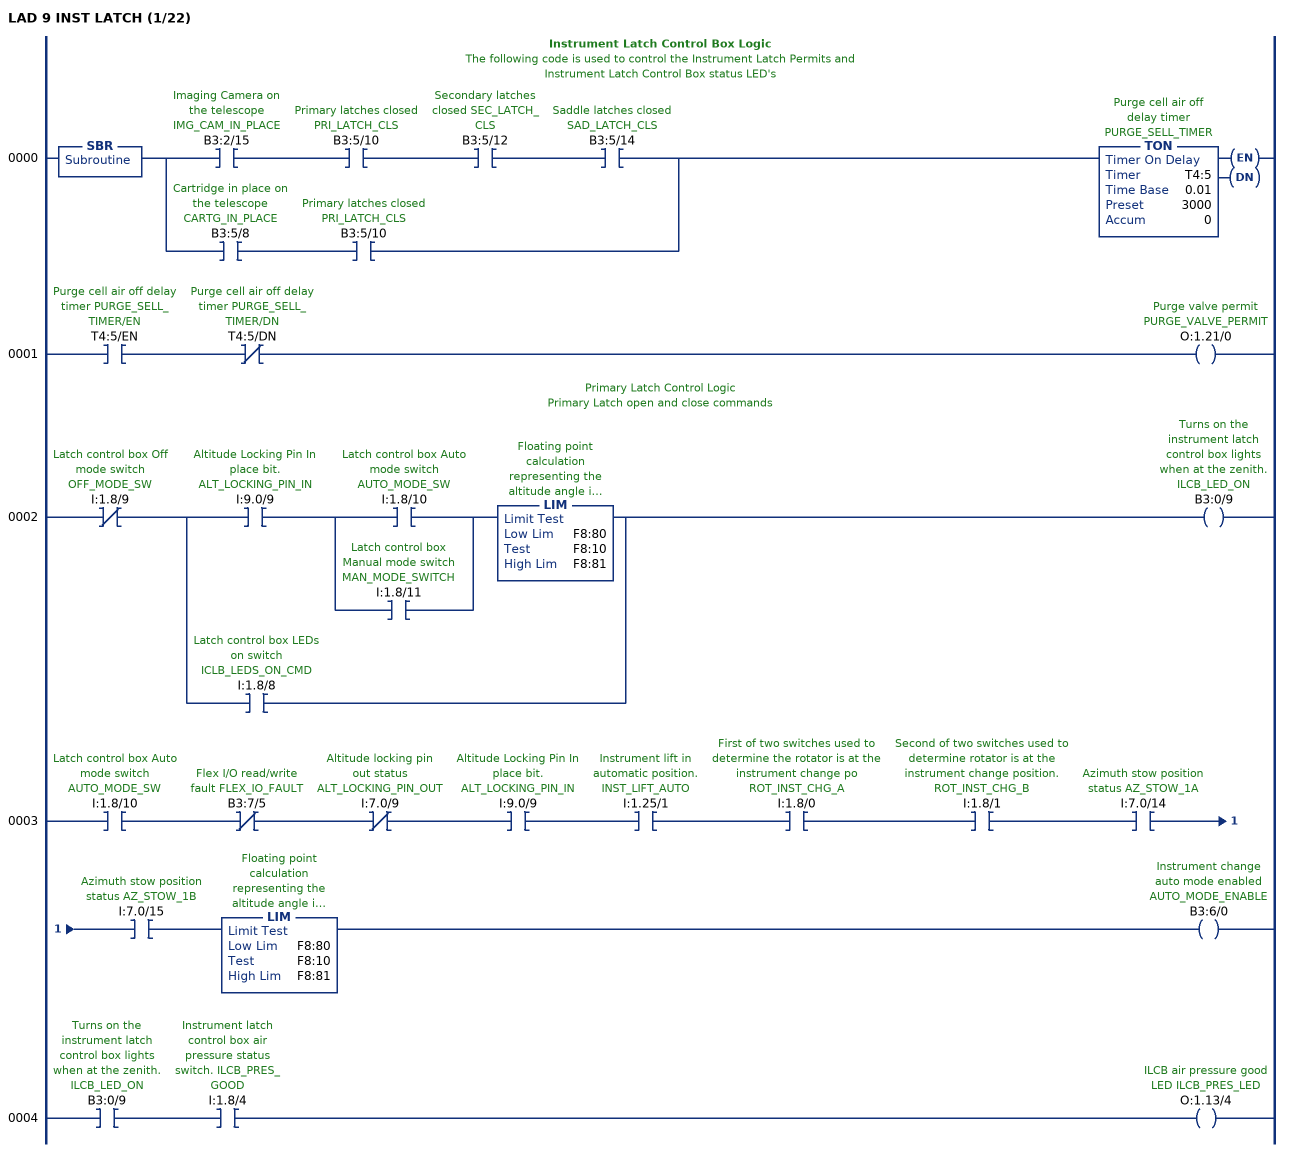
% Rung: 0 %
% TITLE: Instrument Latch Control Box Logic %
% The following code is used to control the Instrument Latch Permits and
% Instrument Latch Control Box status LED's %
SOR SBR BST XIC B3:2/15 XIC B3:5/10 XIC B3:5/12 XIC B3:5/14 NXB XIC B3:5/8 XIC B3:5/10 BND TON T4:5 0.01 3000 0 EOR
%   B3:2/15  IMG_CAM_IN_PLACE  "Imaging Camera on the telescope" %
%   B3:5/10  PRI_LATCH_CLS  "Primary latches closed" %
%   B3:5/12  SEC_LATCH_CLS  "Secondary latches closed" %
%   B3:5/14  SAD_LATCH_CLS  "Saddle latches closed" %
%   B3:5/8  CARTG_IN_PLACE  "Cartridge in place on the telescope" %
%   T4:5  PURGE_SELL_TIMER  "Purge cell air off delay timer" %
% Rung: 1 %
SOR XIC T4:5/EN XIO T4:5/DN OTE O:1.21/0 EOR
%   T4:5  PURGE_SELL_TIMER  "Purge cell air off delay timer" %
%   O:1.21/0  PURGE_VALVE_PERMIT  "Purge valve permit" %
% Rung: 2 %
% Primary Latch Control Logic
% 
% 
% 
% Primary Latch open and close commands %
SOR XIO I:1.8/9 BST XIC I:9.0/9 BST XIC I:1.8/10 NXB XIC I:1.8/11 BND LIM F8:80 F8:10 F8:81 NXB XIC I:1.8/8 BND OTE B3:0/9 EOR
%   I:1.8/9  OFF_MODE_SW  "Latch control box Off mode switch" %
%   I:9.0/9  ALT_LOCKING_PIN_IN  "Altitude Locking Pin In place bit." %
%   I:1.8/10  AUTO_MODE_SW  "Latch control box Auto mode switch" %
%   I:1.8/11  MAN_MODE_SWITCH  "Latch control box Manual mode switch" %
%   F8:80  INST_CHG_LOW_LMT  "The Lower altitude limit to allow instrument change operations" %
%   F8:10  ALT_ANGLE  "Floating point calculation representing the altitude angle in degrees." %
%   F8:81  INST_CHG_HIGH_LMT  "The Upper altitude limit to allow instrument change operations" %
%   I:1.8/8  ICLB_LEDS_ON_CMD  "Latch control box LEDs on switch" %
%   B3:0/9  ILCB_LED_ON  "Turns on the instrument latch control box lights when at the zenith." %
% Rung: 3 %
SOR XIC I:1.8/10 XIO B3:7/5 XIO I:7.0/9 XIC I:9.0/9 XIC I:1.25/1 XIC I:1.8/0 XIC I:1.8/1 XIC I:7.0/14 XIC I:7.0/15 LIM F8:80 F8:10 F8:81 OTE B3:6/0 EOR
%   I:1.8/10  AUTO_MODE_SW  "Latch control box Auto mode switch" %
%   B3:7/5  FLEX_IO_FAULT  "Flex I/O read/write fault" %
%   I:7.0/9  ALT_LOCKING_PIN_OUT  "Altitude locking pin out status" %
%   I:9.0/9  ALT_LOCKING_PIN_IN  "Altitude Locking Pin In place bit." %
%   I:1.25/1  INST_LIFT_AUTO  "Instrument lift in automatic position." %
%   I:1.8/0  ROT_INST_CHG_A  "First of two switches used to determine the rotator is at the instrument change po" %
%   I:1.8/1  ROT_INST_CHG_B  "Second of two switches used to determine rotator is at the instrument change position." %
%   I:7.0/14  AZ_STOW_1A  "Azimuth stow position status" %
%   I:7.0/15  AZ_STOW_1B  "Azimuth stow position status" %
%   F8:80  INST_CHG_LOW_LMT  "The Lower altitude limit to allow instrument change operations" %
%   F8:10  ALT_ANGLE  "Floating point calculation representing the altitude angle in degrees." %
%   F8:81  INST_CHG_HIGH_LMT  "The Upper altitude limit to allow instrument change operations" %
%   B3:6/0  AUTO_MODE_ENABLE  "Instrument change auto mode enabled" %
% Rung: 4 %
SOR XIC B3:0/9 XIC I:1.8/4 OTE O:1.13/4 EOR
%   B3:0/9  ILCB_LED_ON  "Turns on the instrument latch control box lights when at the zenith." %
%   I:1.8/4  ILCB_PRES_GOOD  "Instrument latch control box air pressure status switch." %
%   O:1.13/4  ILCB_PRES_LED  "ILCB air pressure good LED" %

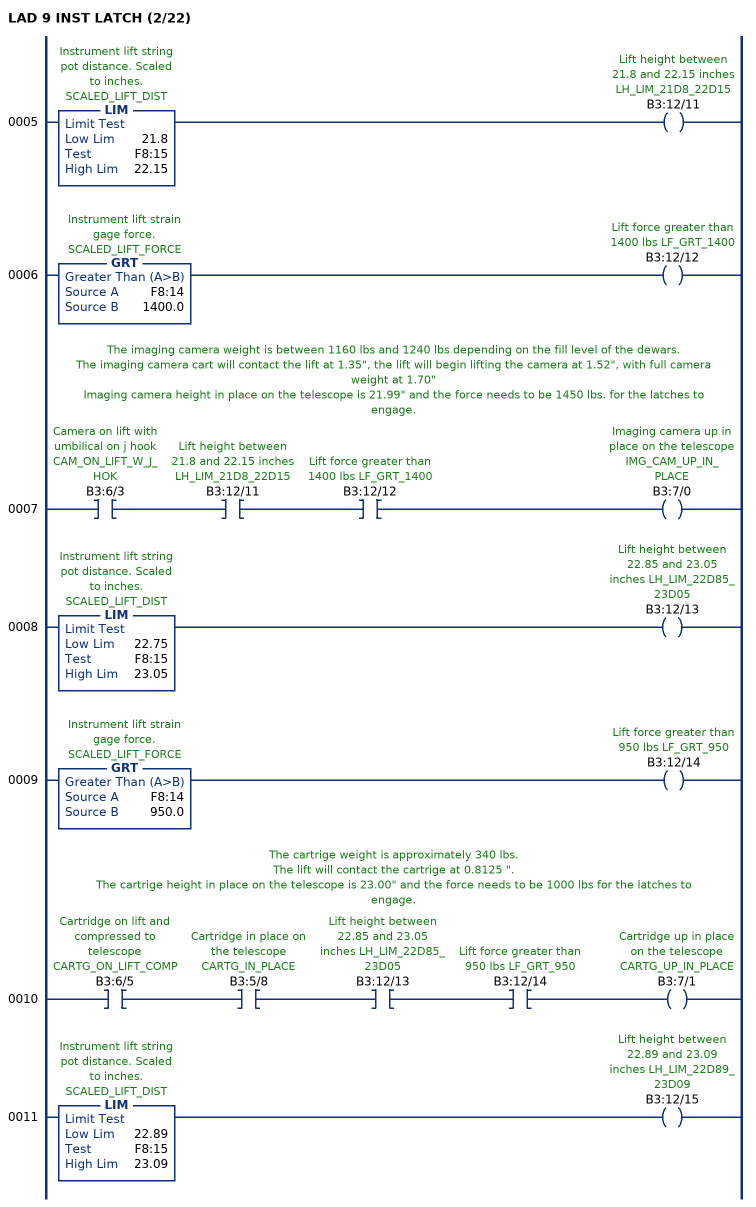
% Rung: 5 %
SOR LIM 21.8 F8:15 22.15 OTE B3:12/11 EOR
%   F8:15  SCALED_LIFT_DIST  "Instrument lift string pot distance. Scaled to inches." %
%   B3:12/11  LH_LIM_21D8_22D15  "Lift height between 21.8 and 22.15 inches" %
% Rung: 6 %
SOR GRT F8:14 1400.0 OTE B3:12/12 EOR
%   F8:14  SCALED_LIFT_FORCE  "Instrument lift strain gage force." %
%   B3:12/12  LF_GRT_1400  "Lift force greater than 1400 lbs" %
% Rung: 7 %
% The imaging camera weight is between 1160 lbs and 1240 lbs depending on the fill level of the dewars.
% The imaging camera cart will contact the lift at 1.35", the lift will begin lifting the camera at 1.52", with full camera weight at 1.70"
% Imaging camera height in place on the telescope is 21.99" and the force needs to be 1450 lbs. for the latches to engage. %
SOR XIC B3:6/3 XIC B3:12/11 XIC B3:12/12 OTE B3:7/0 EOR
%   B3:6/3  CAM_ON_LIFT_W_J_HOK  "Camera on lift with umbilical on j hook" %
%   B3:12/11  LH_LIM_21D8_22D15  "Lift height between 21.8 and 22.15 inches" %
%   B3:12/12  LF_GRT_1400  "Lift force greater than 1400 lbs" %
%   B3:7/0  IMG_CAM_UP_IN_PLACE  "Imaging camera up in place on the telescope" %
% Rung: 8 %
SOR LIM 22.75 F8:15 23.05 OTE B3:12/13 EOR
%   F8:15  SCALED_LIFT_DIST  "Instrument lift string pot distance. Scaled to inches." %
%   B3:12/13  LH_LIM_22D85_23D05  "Lift height between 22.85 and 23.05 inches" %
% Rung: 9 %
SOR GRT F8:14 950.0 OTE B3:12/14 EOR
%   F8:14  SCALED_LIFT_FORCE  "Instrument lift strain gage force." %
%   B3:12/14  LF_GRT_950  "Lift force greater than 950 lbs" %
% Rung: 10 %
% The cartrige weight is approximately 340 lbs.
% The lift will contact the cartrige at 0.8125 ".
% The cartrige height in place on the telescope is 23.00" and the force needs to be 1000 lbs for the latches to engage. %
SOR XIC B3:6/5 XIC B3:5/8 XIC B3:12/13 XIC B3:12/14 OTE B3:7/1 EOR
%   B3:6/5  CARTG_ON_LIFT_COMP  "Cartridge on lift and compressed to telescope" %
%   B3:5/8  CARTG_IN_PLACE  "Cartridge in place on the telescope" %
%   B3:12/13  LH_LIM_22D85_23D05  "Lift height between 22.85 and 23.05 inches" %
%   B3:12/14  LF_GRT_950  "Lift force greater than 950 lbs" %
%   B3:7/1  CARTG_UP_IN_PLACE  "Cartridge up in place on the telescope" %
% Rung: 11 %
SOR LIM 22.89 F8:15 23.09 OTE B3:12/15 EOR
%   F8:15  SCALED_LIFT_DIST  "Instrument lift string pot distance. Scaled to inches." %
%   B3:12/15  LH_LIM_22D89_23D09  "Lift height between 22.89 and 23.09 inches" %

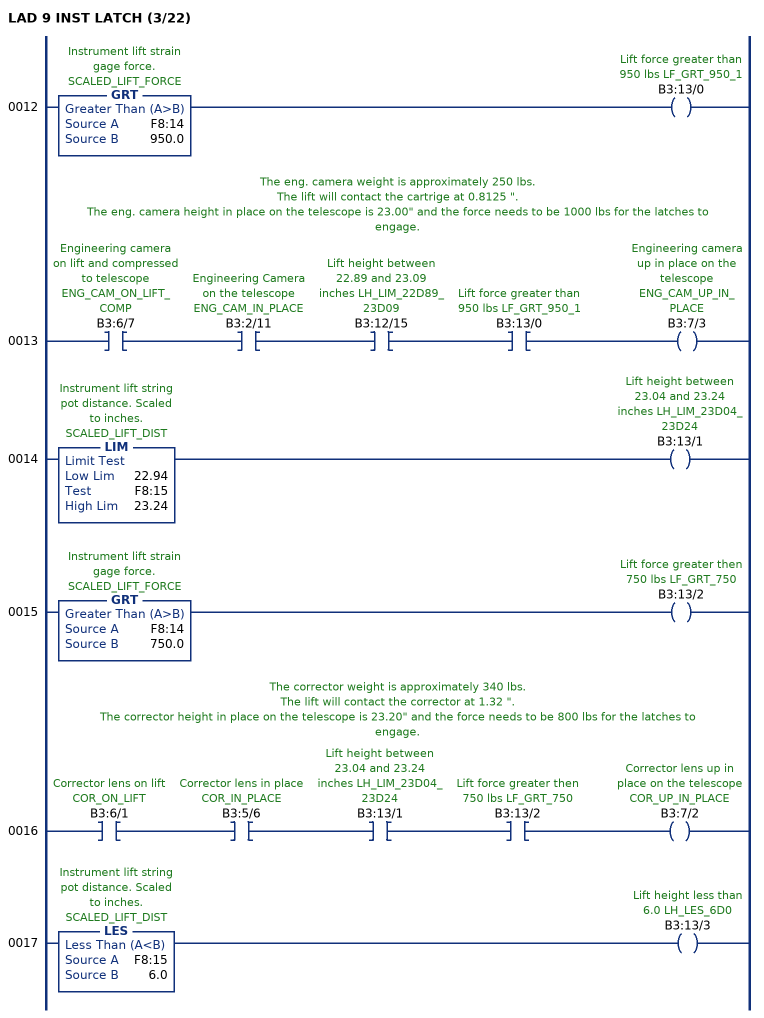
% Rung: 12 %
SOR GRT F8:14 950.0 OTE B3:13/0 EOR
%   F8:14  SCALED_LIFT_FORCE  "Instrument lift strain gage force." %
%   B3:13/0  LF_GRT_950_1  "Lift force greater than 950 lbs" %
% Rung: 13 %
% The eng. camera weight is approximately 250 lbs.
% The lift will contact the cartrige at 0.8125 ".
% The eng. camera height in place on the telescope is 23.00" and the force needs to be 1000 lbs for the latches to engage. %
SOR XIC B3:6/7 XIC B3:2/11 XIC B3:12/15 XIC B3:13/0 OTE B3:7/3 EOR
%   B3:6/7  ENG_CAM_ON_LIFT_COMP  "Engineering camera on lift and compressed to telescope" %
%   B3:2/11  ENG_CAM_IN_PLACE  "Engineering Camera on the telescope" %
%   B3:12/15  LH_LIM_22D89_23D09  "Lift height between 22.89 and 23.09 inches" %
%   B3:13/0  LF_GRT_950_1  "Lift force greater than 950 lbs" %
%   B3:7/3  ENG_CAM_UP_IN_PLACE  "Engineering camera up in place on the telescope" %
% Rung: 14 %
SOR LIM 22.94 F8:15 23.24 OTE B3:13/1 EOR
%   F8:15  SCALED_LIFT_DIST  "Instrument lift string pot distance. Scaled to inches." %
%   B3:13/1  LH_LIM_23D04_23D24  "Lift height between 23.04 and 23.24 inches" %
% Rung: 15 %
SOR GRT F8:14 750.0 OTE B3:13/2 EOR
%   F8:14  SCALED_LIFT_FORCE  "Instrument lift strain gage force." %
%   B3:13/2  LF_GRT_750  "Lift force greater then 750 lbs" %
% Rung: 16 %
% The corrector weight is approximately 340 lbs.
% The lift will contact the corrector at 1.32 ".
% The corrector height in place on the telescope is 23.20" and the force needs to be 800 lbs for the latches to engage. %
SOR XIC B3:6/1 XIC B3:5/6 XIC B3:13/1 XIC B3:13/2 OTE B3:7/2 EOR
%   B3:6/1  COR_ON_LIFT  "Corrector lens on lift" %
%   B3:5/6  COR_IN_PLACE  "Corrector lens in place" %
%   B3:13/1  LH_LIM_23D04_23D24  "Lift height between 23.04 and 23.24 inches" %
%   B3:13/2  LF_GRT_750  "Lift force greater then 750 lbs" %
%   B3:7/2  COR_UP_IN_PLACE  "Corrector lens up in place on the telescope" %
% Rung: 17 %
SOR LES F8:15 6.0 OTE B3:13/3 EOR
%   F8:15  SCALED_LIFT_DIST  "Instrument lift string pot distance. Scaled to inches." %
%   B3:13/3  LH_LES_6D0  "Lift height less than 6.0" %

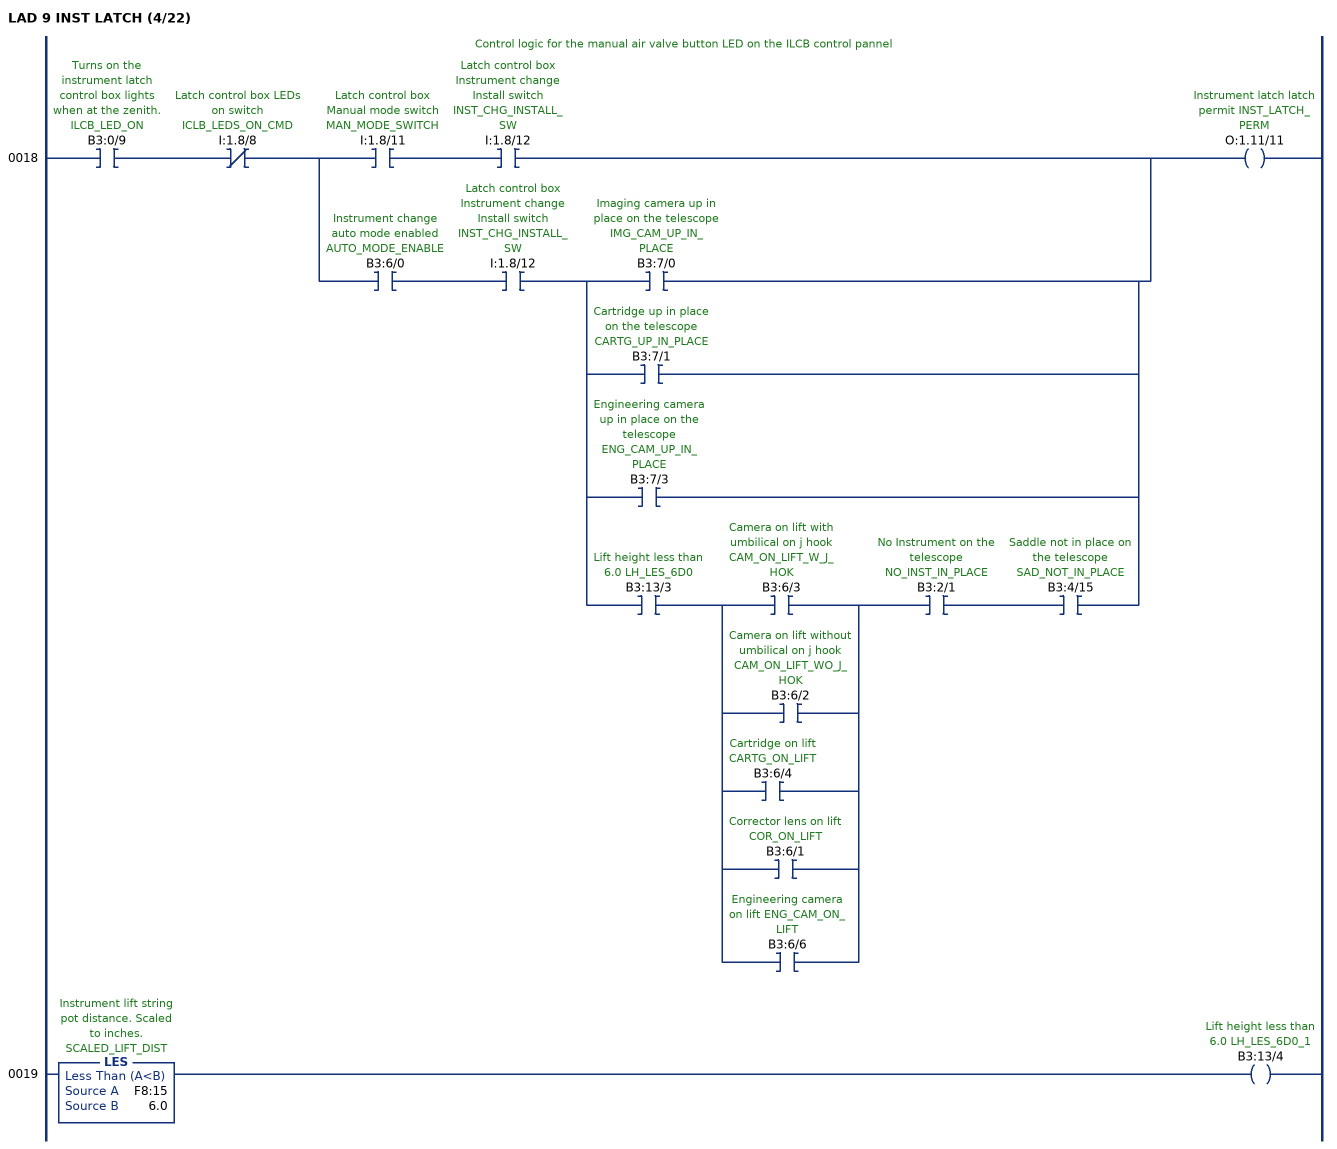
% Rung: 18 %
% Control logic for the manual air valve button LED on the ILCB control pannel %
SOR XIC B3:0/9 XIO I:1.8/8 BST XIC I:1.8/11 XIC I:1.8/12 NXB XIC B3:6/0 XIC I:1.8/12 BST XIC B3:7/0 NXB XIC B3:7/1 NXB XIC B3:7/3 NXB XIC B3:13/3 BST XIC B3:6/3 NXB XIC B3:6/2 NXB XIC B3:6/4 NXB XIC B3:6/1 NXB XIC B3:6/6 BND XIC B3:2/1 XIC B3:4/15 BND BND OTE O:1.11/11 EOR
%   B3:0/9  ILCB_LED_ON  "Turns on the instrument latch control box lights when at the zenith." %
%   I:1.8/8  ICLB_LEDS_ON_CMD  "Latch control box LEDs on switch" %
%   I:1.8/11  MAN_MODE_SWITCH  "Latch control box Manual mode switch" %
%   I:1.8/12  INST_CHG_INSTALL_SW  "Latch control box Instrument change Install switch" %
%   B3:6/0  AUTO_MODE_ENABLE  "Instrument change auto mode enabled" %
%   B3:7/0  IMG_CAM_UP_IN_PLACE  "Imaging camera up in place on the telescope" %
%   B3:7/1  CARTG_UP_IN_PLACE  "Cartridge up in place on the telescope" %
%   B3:7/3  ENG_CAM_UP_IN_PLACE  "Engineering camera up in place on the telescope" %
%   B3:13/3  LH_LES_6D0  "Lift height less than 6.0" %
%   B3:6/3  CAM_ON_LIFT_W_J_HOK  "Camera on lift with umbilical on j hook" %
%   B3:6/2  CAM_ON_LIFT_WO_J_HOK  "Camera on lift without umbilical on j hook" %
%   B3:6/4  CARTG_ON_LIFT  "Cartridge on lift" %
%   B3:6/1  COR_ON_LIFT  "Corrector lens on lift" %
%   B3:6/6  ENG_CAM_ON_LIFT  "Engineering camera on lift" %
%   B3:2/1  NO_INST_IN_PLACE  "No Instrument on the telescope" %
%   B3:4/15  SAD_NOT_IN_PLACE  "Saddle not in place on the telescope" %
%   O:1.11/11  INST_LATCH_PERM  "Instrument latch latch permit" %
% Rung: 19 %
SOR LES F8:15 6.0 OTE B3:13/4 EOR
%   F8:15  SCALED_LIFT_DIST  "Instrument lift string pot distance. Scaled to inches." %
%   B3:13/4  LH_LES_6D0_1  "Lift height less than 6.0" %

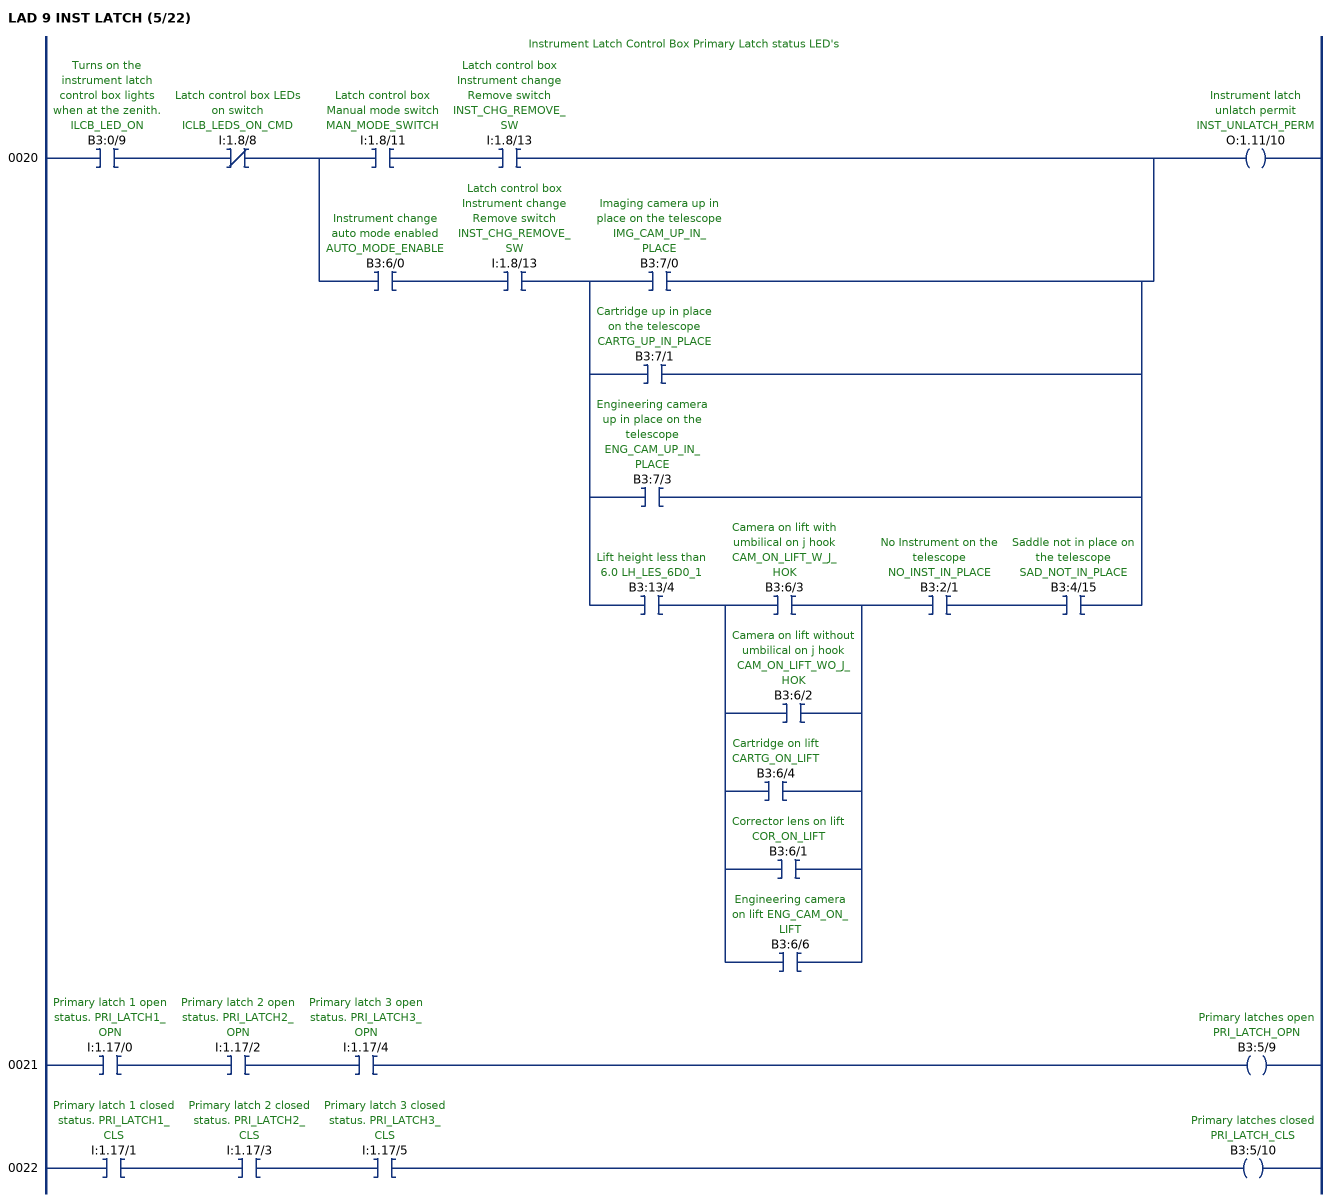
% Rung: 20 %
% Instrument Latch Control Box Primary Latch status LED's %
SOR XIC B3:0/9 XIO I:1.8/8 BST XIC I:1.8/11 XIC I:1.8/13 NXB XIC B3:6/0 XIC I:1.8/13 BST XIC B3:7/0 NXB XIC B3:7/1 NXB XIC B3:7/3 NXB XIC B3:13/4 BST XIC B3:6/3 NXB XIC B3:6/2 NXB XIC B3:6/4 NXB XIC B3:6/1 NXB XIC B3:6/6 BND XIC B3:2/1 XIC B3:4/15 BND BND OTE O:1.11/10 EOR
%   B3:0/9  ILCB_LED_ON  "Turns on the instrument latch control box lights when at the zenith." %
%   I:1.8/8  ICLB_LEDS_ON_CMD  "Latch control box LEDs on switch" %
%   I:1.8/11  MAN_MODE_SWITCH  "Latch control box Manual mode switch" %
%   I:1.8/13  INST_CHG_REMOVE_SW  "Latch control box Instrument change Remove switch" %
%   B3:6/0  AUTO_MODE_ENABLE  "Instrument change auto mode enabled" %
%   B3:7/0  IMG_CAM_UP_IN_PLACE  "Imaging camera up in place on the telescope" %
%   B3:7/1  CARTG_UP_IN_PLACE  "Cartridge up in place on the telescope" %
%   B3:7/3  ENG_CAM_UP_IN_PLACE  "Engineering camera up in place on the telescope" %
%   B3:13/4  LH_LES_6D0_1  "Lift height less than 6.0" %
%   B3:6/3  CAM_ON_LIFT_W_J_HOK  "Camera on lift with umbilical on j hook" %
%   B3:6/2  CAM_ON_LIFT_WO_J_HOK  "Camera on lift without umbilical on j hook" %
%   B3:6/4  CARTG_ON_LIFT  "Cartridge on lift" %
%   B3:6/1  COR_ON_LIFT  "Corrector lens on lift" %
%   B3:6/6  ENG_CAM_ON_LIFT  "Engineering camera on lift" %
%   B3:2/1  NO_INST_IN_PLACE  "No Instrument on the telescope" %
%   B3:4/15  SAD_NOT_IN_PLACE  "Saddle not in place on the telescope" %
%   O:1.11/10  INST_UNLATCH_PERM  "Instrument latch unlatch permit" %
% Rung: 21 %
SOR XIC I:1.17/0 XIC I:1.17/2 XIC I:1.17/4 OTE B3:5/9 EOR
%   I:1.17/0  PRI_LATCH1_OPN  "Primary latch 1 open status." %
%   I:1.17/2  PRI_LATCH2_OPN  "Primary latch 2 open status." %
%   I:1.17/4  PRI_LATCH3_OPN  "Primary latch 3 open status." %
%   B3:5/9  PRI_LATCH_OPN  "Primary latches open" %
% Rung: 22 %
SOR XIC I:1.17/1 XIC I:1.17/3 XIC I:1.17/5 OTE B3:5/10 EOR
%   I:1.17/1  PRI_LATCH1_CLS  "Primary latch 1 closed status." %
%   I:1.17/3  PRI_LATCH2_CLS  "Primary latch 2 closed status." %
%   I:1.17/5  PRI_LATCH3_CLS  "Primary latch 3 closed status." %
%   B3:5/10  PRI_LATCH_CLS  "Primary latches closed" %

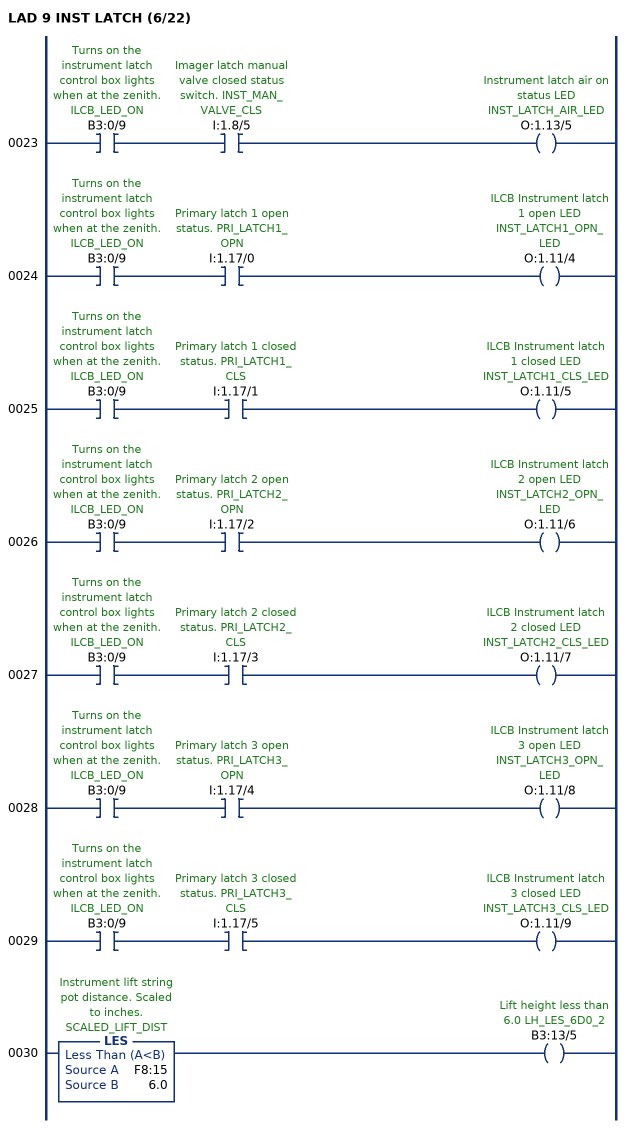
% Rung: 23 %
SOR XIC B3:0/9 XIC I:1.8/5 OTE O:1.13/5 EOR
%   B3:0/9  ILCB_LED_ON  "Turns on the instrument latch control box lights when at the zenith." %
%   I:1.8/5  INST_MAN_VALVE_CLS  "Imager latch manual valve closed status switch." %
%   O:1.13/5  INST_LATCH_AIR_LED  "Instrument latch air on status LED" %
% Rung: 24 %
SOR XIC B3:0/9 XIC I:1.17/0 OTE O:1.11/4 EOR
%   B3:0/9  ILCB_LED_ON  "Turns on the instrument latch control box lights when at the zenith." %
%   I:1.17/0  PRI_LATCH1_OPN  "Primary latch 1 open status." %
%   O:1.11/4  INST_LATCH1_OPN_LED  "ILCB Instrument latch 1 open LED" %
% Rung: 25 %
SOR XIC B3:0/9 XIC I:1.17/1 OTE O:1.11/5 EOR
%   B3:0/9  ILCB_LED_ON  "Turns on the instrument latch control box lights when at the zenith." %
%   I:1.17/1  PRI_LATCH1_CLS  "Primary latch 1 closed status." %
%   O:1.11/5  INST_LATCH1_CLS_LED  "ILCB Instrument latch 1 closed LED" %
% Rung: 26 %
SOR XIC B3:0/9 XIC I:1.17/2 OTE O:1.11/6 EOR
%   B3:0/9  ILCB_LED_ON  "Turns on the instrument latch control box lights when at the zenith." %
%   I:1.17/2  PRI_LATCH2_OPN  "Primary latch 2 open status." %
%   O:1.11/6  INST_LATCH2_OPN_LED  "ILCB Instrument latch 2 open LED" %
% Rung: 27 %
SOR XIC B3:0/9 XIC I:1.17/3 OTE O:1.11/7 EOR
%   B3:0/9  ILCB_LED_ON  "Turns on the instrument latch control box lights when at the zenith." %
%   I:1.17/3  PRI_LATCH2_CLS  "Primary latch 2 closed status." %
%   O:1.11/7  INST_LATCH2_CLS_LED  "ILCB Instrument latch 2 closed LED" %
% Rung: 28 %
SOR XIC B3:0/9 XIC I:1.17/4 OTE O:1.11/8 EOR
%   B3:0/9  ILCB_LED_ON  "Turns on the instrument latch control box lights when at the zenith." %
%   I:1.17/4  PRI_LATCH3_OPN  "Primary latch 3 open status." %
%   O:1.11/8  INST_LATCH3_OPN_LED  "ILCB Instrument latch 3 open LED" %
% Rung: 29 %
SOR XIC B3:0/9 XIC I:1.17/5 OTE O:1.11/9 EOR
%   B3:0/9  ILCB_LED_ON  "Turns on the instrument latch control box lights when at the zenith." %
%   I:1.17/5  PRI_LATCH3_CLS  "Primary latch 3 closed status." %
%   O:1.11/9  INST_LATCH3_CLS_LED  "ILCB Instrument latch 3 closed LED" %
% Rung: 30 %
SOR LES F8:15 6.0 OTE B3:13/5 EOR
%   F8:15  SCALED_LIFT_DIST  "Instrument lift string pot distance. Scaled to inches." %
%   B3:13/5  LH_LES_6D0_2  "Lift height less than 6.0" %

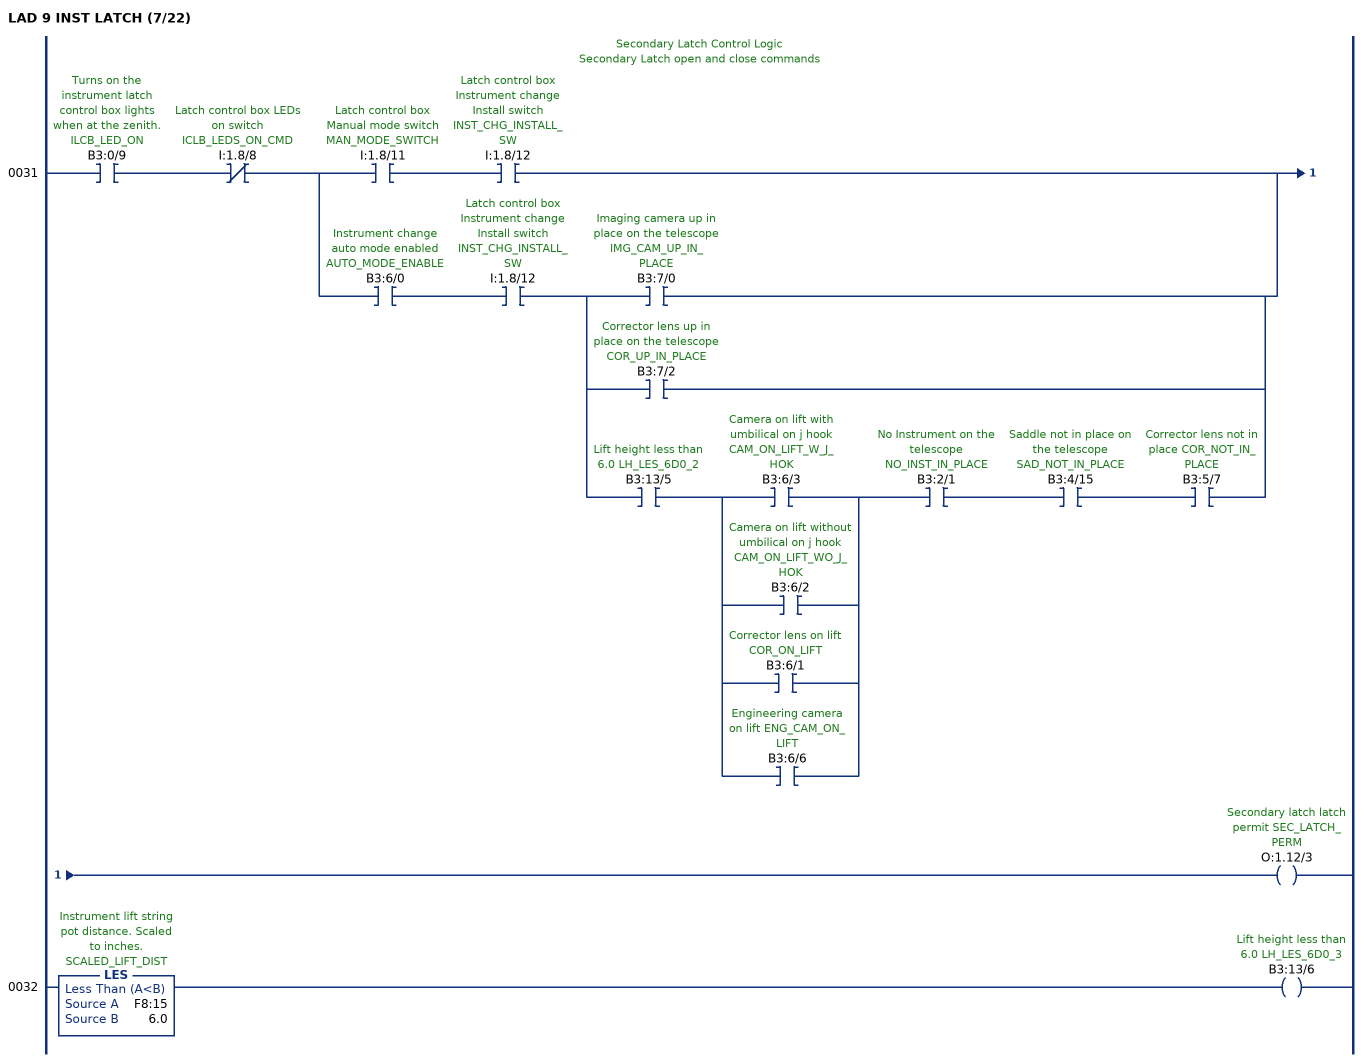
% Rung: 31 %
% Secondary Latch Control Logic
% 
% 
% 
% Secondary Latch open and close commands %
SOR XIC B3:0/9 XIO I:1.8/8 BST XIC I:1.8/11 XIC I:1.8/12 NXB XIC B3:6/0 XIC I:1.8/12 BST XIC B3:7/0 NXB XIC B3:7/2 NXB XIC B3:13/5 BST XIC B3:6/3 NXB XIC B3:6/2 NXB XIC B3:6/1 NXB XIC B3:6/6 BND XIC B3:2/1 XIC B3:4/15 XIC B3:5/7 BND BND OTE O:1.12/3 EOR
%   B3:0/9  ILCB_LED_ON  "Turns on the instrument latch control box lights when at the zenith." %
%   I:1.8/8  ICLB_LEDS_ON_CMD  "Latch control box LEDs on switch" %
%   I:1.8/11  MAN_MODE_SWITCH  "Latch control box Manual mode switch" %
%   I:1.8/12  INST_CHG_INSTALL_SW  "Latch control box Instrument change Install switch" %
%   B3:6/0  AUTO_MODE_ENABLE  "Instrument change auto mode enabled" %
%   B3:7/0  IMG_CAM_UP_IN_PLACE  "Imaging camera up in place on the telescope" %
%   B3:7/2  COR_UP_IN_PLACE  "Corrector lens up in place on the telescope" %
%   B3:13/5  LH_LES_6D0_2  "Lift height less than 6.0" %
%   B3:6/3  CAM_ON_LIFT_W_J_HOK  "Camera on lift with umbilical on j hook" %
%   B3:6/2  CAM_ON_LIFT_WO_J_HOK  "Camera on lift without umbilical on j hook" %
%   B3:6/1  COR_ON_LIFT  "Corrector lens on lift" %
%   B3:6/6  ENG_CAM_ON_LIFT  "Engineering camera on lift" %
%   B3:2/1  NO_INST_IN_PLACE  "No Instrument on the telescope" %
%   B3:4/15  SAD_NOT_IN_PLACE  "Saddle not in place on the telescope" %
%   B3:5/7  COR_NOT_IN_PLACE  "Corrector lens not in place" %
%   O:1.12/3  SEC_LATCH_PERM  "Secondary latch latch permit" %
% Rung: 32 %
SOR LES F8:15 6.0 OTE B3:13/6 EOR
%   F8:15  SCALED_LIFT_DIST  "Instrument lift string pot distance. Scaled to inches." %
%   B3:13/6  LH_LES_6D0_3  "Lift height less than 6.0" %

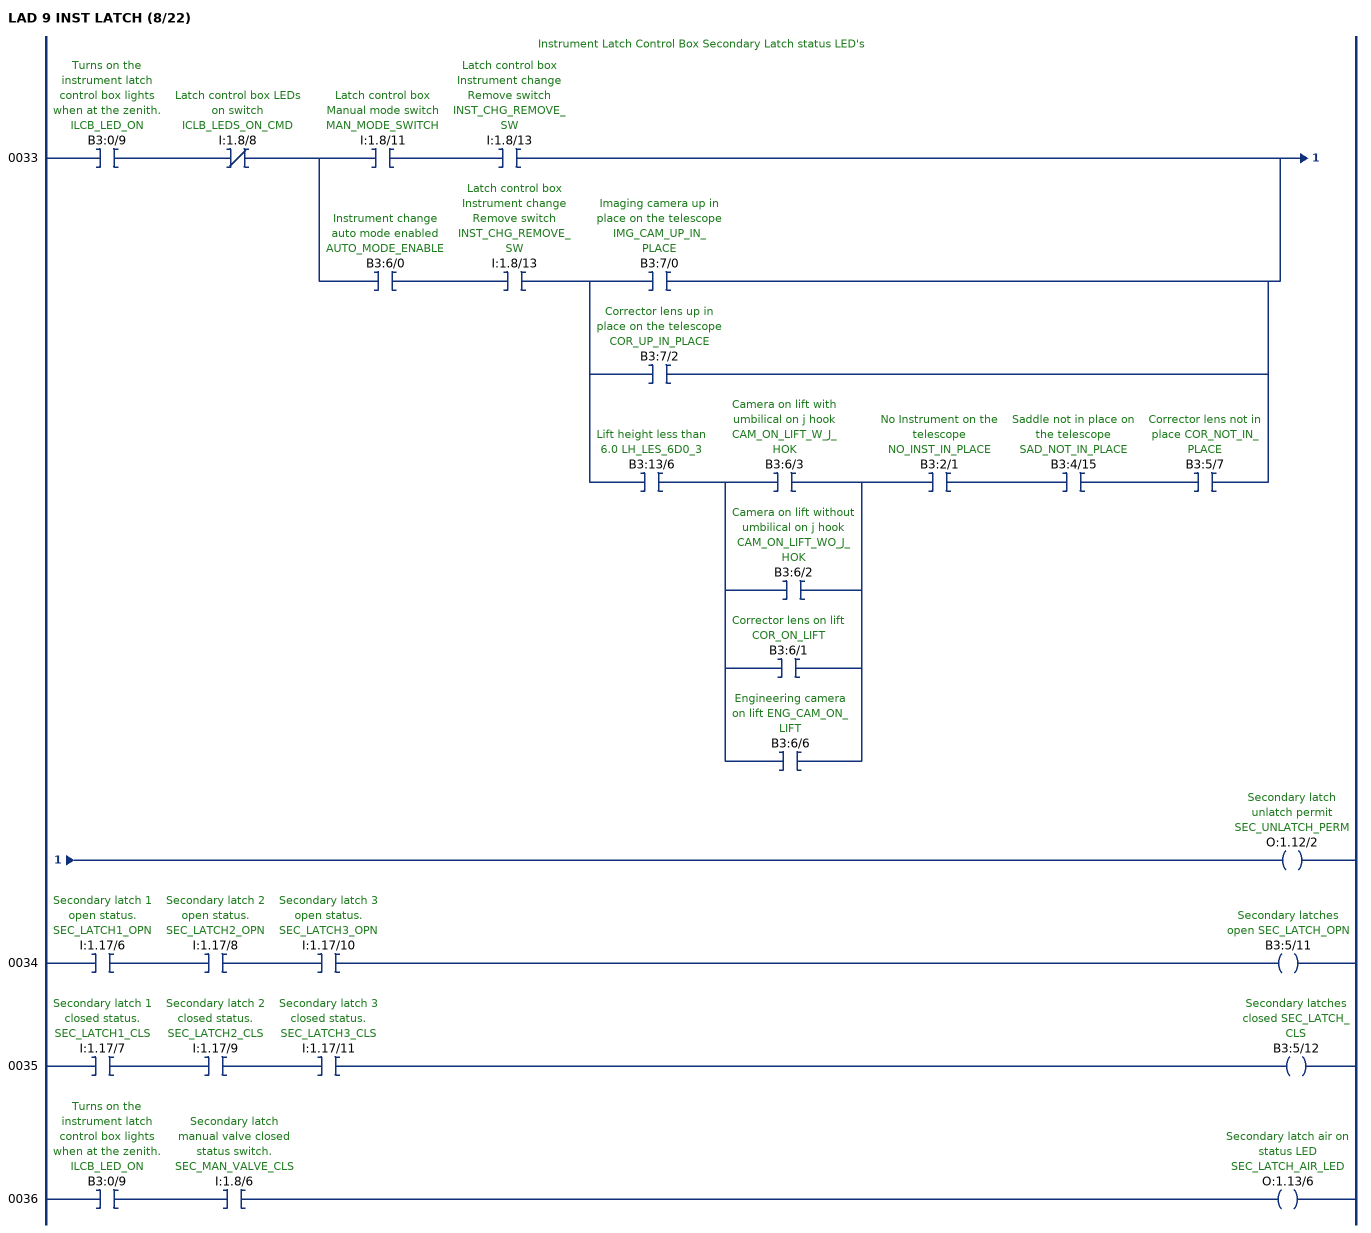
% Rung: 33 %
% Instrument Latch Control Box Secondary Latch status LED's %
SOR XIC B3:0/9 XIO I:1.8/8 BST XIC I:1.8/11 XIC I:1.8/13 NXB XIC B3:6/0 XIC I:1.8/13 BST XIC B3:7/0 NXB XIC B3:7/2 NXB XIC B3:13/6 BST XIC B3:6/3 NXB XIC B3:6/2 NXB XIC B3:6/1 NXB XIC B3:6/6 BND XIC B3:2/1 XIC B3:4/15 XIC B3:5/7 BND BND OTE O:1.12/2 EOR
%   B3:0/9  ILCB_LED_ON  "Turns on the instrument latch control box lights when at the zenith." %
%   I:1.8/8  ICLB_LEDS_ON_CMD  "Latch control box LEDs on switch" %
%   I:1.8/11  MAN_MODE_SWITCH  "Latch control box Manual mode switch" %
%   I:1.8/13  INST_CHG_REMOVE_SW  "Latch control box Instrument change Remove switch" %
%   B3:6/0  AUTO_MODE_ENABLE  "Instrument change auto mode enabled" %
%   B3:7/0  IMG_CAM_UP_IN_PLACE  "Imaging camera up in place on the telescope" %
%   B3:7/2  COR_UP_IN_PLACE  "Corrector lens up in place on the telescope" %
%   B3:13/6  LH_LES_6D0_3  "Lift height less than 6.0" %
%   B3:6/3  CAM_ON_LIFT_W_J_HOK  "Camera on lift with umbilical on j hook" %
%   B3:6/2  CAM_ON_LIFT_WO_J_HOK  "Camera on lift without umbilical on j hook" %
%   B3:6/1  COR_ON_LIFT  "Corrector lens on lift" %
%   B3:6/6  ENG_CAM_ON_LIFT  "Engineering camera on lift" %
%   B3:2/1  NO_INST_IN_PLACE  "No Instrument on the telescope" %
%   B3:4/15  SAD_NOT_IN_PLACE  "Saddle not in place on the telescope" %
%   B3:5/7  COR_NOT_IN_PLACE  "Corrector lens not in place" %
%   O:1.12/2  SEC_UNLATCH_PERM  "Secondary latch unlatch permit" %
% Rung: 34 %
SOR XIC I:1.17/6 XIC I:1.17/8 XIC I:1.17/10 OTE B3:5/11 EOR
%   I:1.17/6  SEC_LATCH1_OPN  "Secondary latch 1 open status." %
%   I:1.17/8  SEC_LATCH2_OPN  "Secondary latch 2 open status." %
%   I:1.17/10  SEC_LATCH3_OPN  "Secondary latch 3 open status." %
%   B3:5/11  SEC_LATCH_OPN  "Secondary latches open" %
% Rung: 35 %
SOR XIC I:1.17/7 XIC I:1.17/9 XIC I:1.17/11 OTE B3:5/12 EOR
%   I:1.17/7  SEC_LATCH1_CLS  "Secondary latch 1 closed status." %
%   I:1.17/9  SEC_LATCH2_CLS  "Secondary latch 2 closed status." %
%   I:1.17/11  SEC_LATCH3_CLS  "Secondary latch 3 closed status." %
%   B3:5/12  SEC_LATCH_CLS  "Secondary latches closed" %
% Rung: 36 %
SOR XIC B3:0/9 XIC I:1.8/6 OTE O:1.13/6 EOR
%   B3:0/9  ILCB_LED_ON  "Turns on the instrument latch control box lights when at the zenith." %
%   I:1.8/6  SEC_MAN_VALVE_CLS  "Secondary latch manual valve closed status switch." %
%   O:1.13/6  SEC_LATCH_AIR_LED  "Secondary latch air on status LED" %

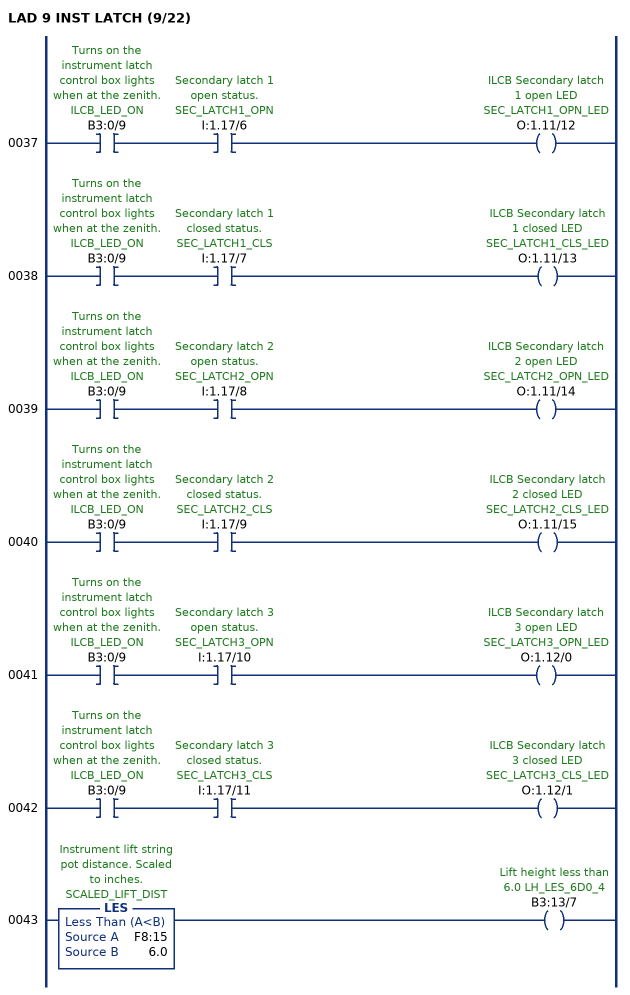
% Rung: 37 %
SOR XIC B3:0/9 XIC I:1.17/6 OTE O:1.11/12 EOR
%   B3:0/9  ILCB_LED_ON  "Turns on the instrument latch control box lights when at the zenith." %
%   I:1.17/6  SEC_LATCH1_OPN  "Secondary latch 1 open status." %
%   O:1.11/12  SEC_LATCH1_OPN_LED  "ILCB Secondary latch 1 open LED" %
% Rung: 38 %
SOR XIC B3:0/9 XIC I:1.17/7 OTE O:1.11/13 EOR
%   B3:0/9  ILCB_LED_ON  "Turns on the instrument latch control box lights when at the zenith." %
%   I:1.17/7  SEC_LATCH1_CLS  "Secondary latch 1 closed status." %
%   O:1.11/13  SEC_LATCH1_CLS_LED  "ILCB Secondary latch 1 closed LED" %
% Rung: 39 %
SOR XIC B3:0/9 XIC I:1.17/8 OTE O:1.11/14 EOR
%   B3:0/9  ILCB_LED_ON  "Turns on the instrument latch control box lights when at the zenith." %
%   I:1.17/8  SEC_LATCH2_OPN  "Secondary latch 2 open status." %
%   O:1.11/14  SEC_LATCH2_OPN_LED  "ILCB Secondary latch 2 open LED" %
% Rung: 40 %
SOR XIC B3:0/9 XIC I:1.17/9 OTE O:1.11/15 EOR
%   B3:0/9  ILCB_LED_ON  "Turns on the instrument latch control box lights when at the zenith." %
%   I:1.17/9  SEC_LATCH2_CLS  "Secondary latch 2 closed status." %
%   O:1.11/15  SEC_LATCH2_CLS_LED  "ILCB Secondary latch 2 closed LED" %
% Rung: 41 %
SOR XIC B3:0/9 XIC I:1.17/10 OTE O:1.12/0 EOR
%   B3:0/9  ILCB_LED_ON  "Turns on the instrument latch control box lights when at the zenith." %
%   I:1.17/10  SEC_LATCH3_OPN  "Secondary latch 3 open status." %
%   O:1.12/0  SEC_LATCH3_OPN_LED  "ILCB Secondary latch 3 open LED" %
% Rung: 42 %
SOR XIC B3:0/9 XIC I:1.17/11 OTE O:1.12/1 EOR
%   B3:0/9  ILCB_LED_ON  "Turns on the instrument latch control box lights when at the zenith." %
%   I:1.17/11  SEC_LATCH3_CLS  "Secondary latch 3 closed status." %
%   O:1.12/1  SEC_LATCH3_CLS_LED  "ILCB Secondary latch 3 closed LED" %
% Rung: 43 %
SOR LES F8:15 6.0 OTE B3:13/7 EOR
%   F8:15  SCALED_LIFT_DIST  "Instrument lift string pot distance. Scaled to inches." %
%   B3:13/7  LH_LES_6D0_4  "Lift height less than 6.0" %

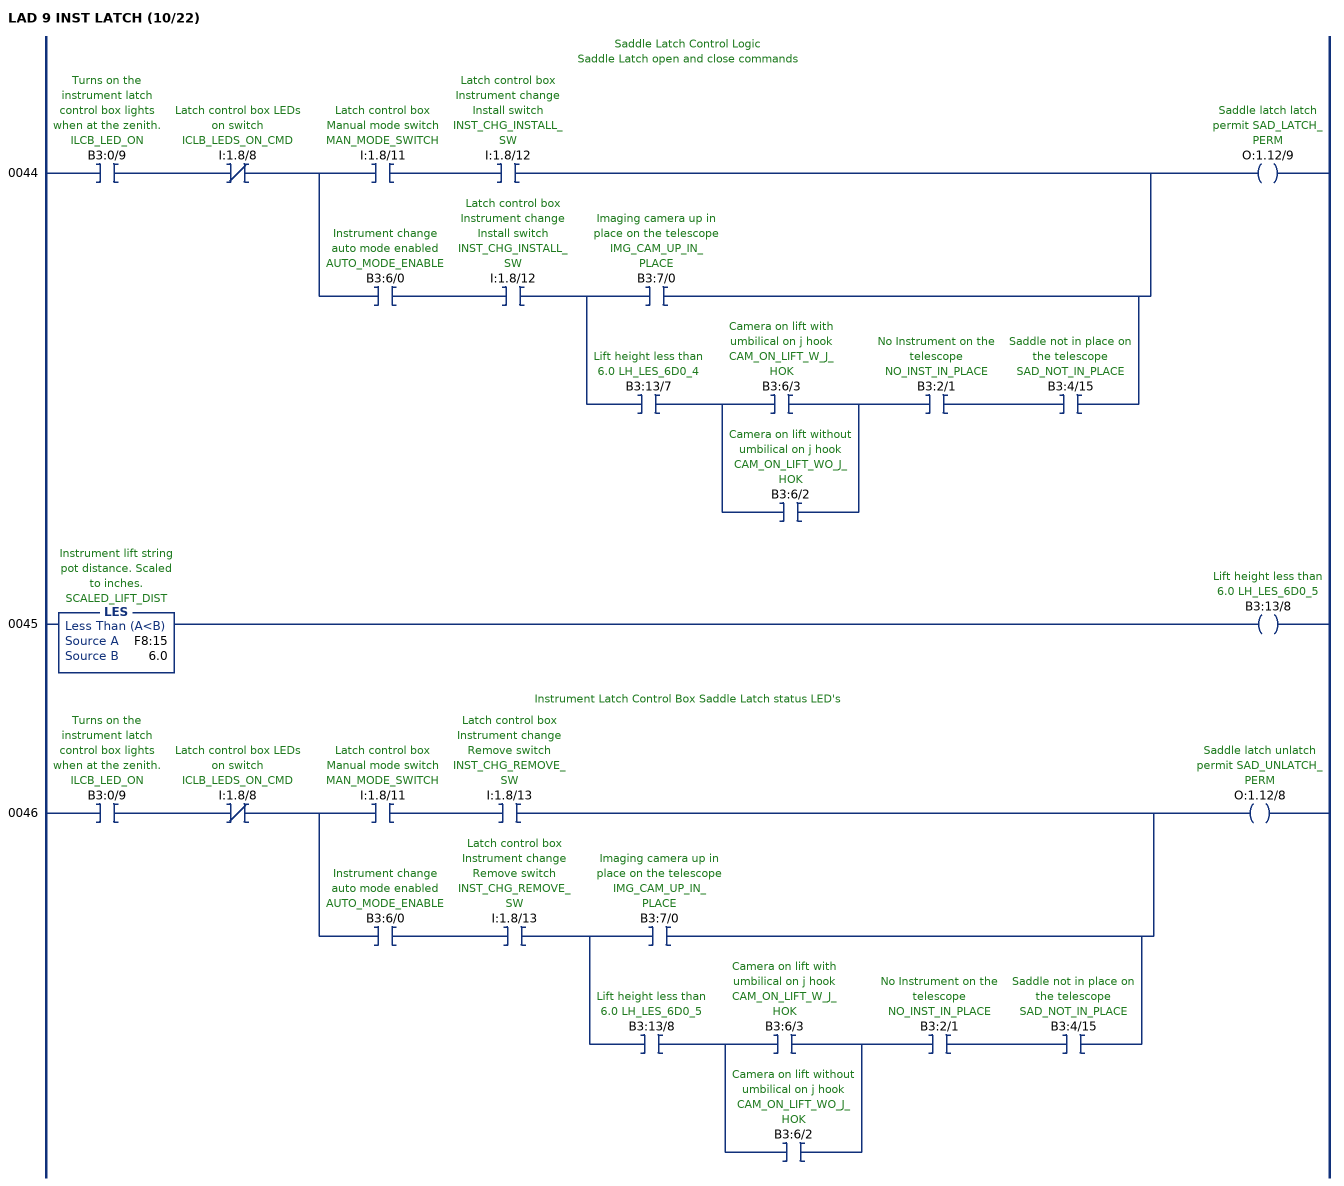
% Rung: 44 %
% Saddle Latch Control Logic
% 
% 
% 
% Saddle Latch open and close commands %
SOR XIC B3:0/9 XIO I:1.8/8 BST XIC I:1.8/11 XIC I:1.8/12 NXB XIC B3:6/0 XIC I:1.8/12 BST XIC B3:7/0 NXB XIC B3:13/7 BST XIC B3:6/3 NXB XIC B3:6/2 BND XIC B3:2/1 XIC B3:4/15 BND BND OTE O:1.12/9 EOR
%   B3:0/9  ILCB_LED_ON  "Turns on the instrument latch control box lights when at the zenith." %
%   I:1.8/8  ICLB_LEDS_ON_CMD  "Latch control box LEDs on switch" %
%   I:1.8/11  MAN_MODE_SWITCH  "Latch control box Manual mode switch" %
%   I:1.8/12  INST_CHG_INSTALL_SW  "Latch control box Instrument change Install switch" %
%   B3:6/0  AUTO_MODE_ENABLE  "Instrument change auto mode enabled" %
%   B3:7/0  IMG_CAM_UP_IN_PLACE  "Imaging camera up in place on the telescope" %
%   B3:13/7  LH_LES_6D0_4  "Lift height less than 6.0" %
%   B3:6/3  CAM_ON_LIFT_W_J_HOK  "Camera on lift with umbilical on j hook" %
%   B3:6/2  CAM_ON_LIFT_WO_J_HOK  "Camera on lift without umbilical on j hook" %
%   B3:2/1  NO_INST_IN_PLACE  "No Instrument on the telescope" %
%   B3:4/15  SAD_NOT_IN_PLACE  "Saddle not in place on the telescope" %
%   O:1.12/9  SAD_LATCH_PERM  "Saddle latch latch permit" %
% Rung: 45 %
SOR LES F8:15 6.0 OTE B3:13/8 EOR
%   F8:15  SCALED_LIFT_DIST  "Instrument lift string pot distance. Scaled to inches." %
%   B3:13/8  LH_LES_6D0_5  "Lift height less than 6.0" %
% Rung: 46 %
% Instrument Latch Control Box Saddle Latch status LED's %
SOR XIC B3:0/9 XIO I:1.8/8 BST XIC I:1.8/11 XIC I:1.8/13 NXB XIC B3:6/0 XIC I:1.8/13 BST XIC B3:7/0 NXB XIC B3:13/8 BST XIC B3:6/3 NXB XIC B3:6/2 BND XIC B3:2/1 XIC B3:4/15 BND BND OTE O:1.12/8 EOR
%   B3:0/9  ILCB_LED_ON  "Turns on the instrument latch control box lights when at the zenith." %
%   I:1.8/8  ICLB_LEDS_ON_CMD  "Latch control box LEDs on switch" %
%   I:1.8/11  MAN_MODE_SWITCH  "Latch control box Manual mode switch" %
%   I:1.8/13  INST_CHG_REMOVE_SW  "Latch control box Instrument change Remove switch" %
%   B3:6/0  AUTO_MODE_ENABLE  "Instrument change auto mode enabled" %
%   B3:7/0  IMG_CAM_UP_IN_PLACE  "Imaging camera up in place on the telescope" %
%   B3:13/8  LH_LES_6D0_5  "Lift height less than 6.0" %
%   B3:6/3  CAM_ON_LIFT_W_J_HOK  "Camera on lift with umbilical on j hook" %
%   B3:6/2  CAM_ON_LIFT_WO_J_HOK  "Camera on lift without umbilical on j hook" %
%   B3:2/1  NO_INST_IN_PLACE  "No Instrument on the telescope" %
%   B3:4/15  SAD_NOT_IN_PLACE  "Saddle not in place on the telescope" %
%   O:1.12/8  SAD_UNLATCH_PERM  "Saddle latch unlatch permit" %

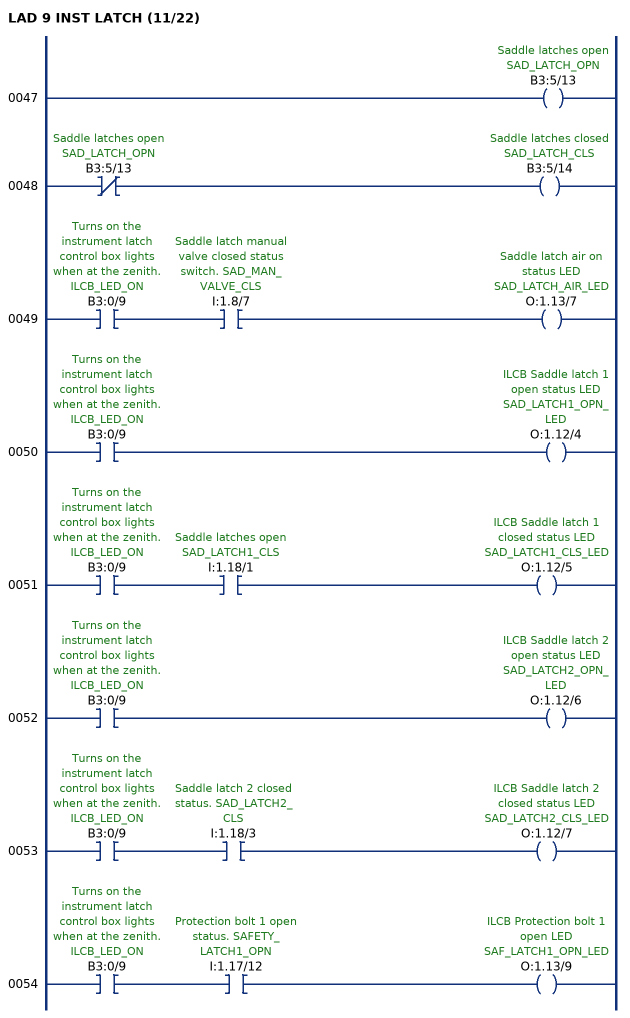
% Rung: 47 %
SOR OTE B3:5/13 EOR
%   B3:5/13  SAD_LATCH_OPN  "Saddle latches open" %
% Rung: 48 %
SOR XIO B3:5/13 OTE B3:5/14 EOR
%   B3:5/13  SAD_LATCH_OPN  "Saddle latches open" %
%   B3:5/14  SAD_LATCH_CLS  "Saddle latches closed" %
% Rung: 49 %
SOR XIC B3:0/9 XIC I:1.8/7 OTE O:1.13/7 EOR
%   B3:0/9  ILCB_LED_ON  "Turns on the instrument latch control box lights when at the zenith." %
%   I:1.8/7  SAD_MAN_VALVE_CLS  "Saddle latch manual valve closed status switch." %
%   O:1.13/7  SAD_LATCH_AIR_LED  "Saddle latch air on status LED" %
% Rung: 50 %
SOR XIC B3:0/9 OTE O:1.12/4 EOR
%   B3:0/9  ILCB_LED_ON  "Turns on the instrument latch control box lights when at the zenith." %
%   O:1.12/4  SAD_LATCH1_OPN_LED  "ILCB Saddle latch 1 open status LED" %
% Rung: 51 %
SOR XIC B3:0/9 XIC I:1.18/1 OTE O:1.12/5 EOR
%   B3:0/9  ILCB_LED_ON  "Turns on the instrument latch control box lights when at the zenith." %
%   I:1.18/1  SAD_LATCH1_CLS  "Saddle latches open" %
%   O:1.12/5  SAD_LATCH1_CLS_LED  "ILCB Saddle latch 1 closed status LED" %
% Rung: 52 %
SOR XIC B3:0/9 OTE O:1.12/6 EOR
%   B3:0/9  ILCB_LED_ON  "Turns on the instrument latch control box lights when at the zenith." %
%   O:1.12/6  SAD_LATCH2_OPN_LED  "ILCB Saddle latch 2 open status LED" %
% Rung: 53 %
SOR XIC B3:0/9 XIC I:1.18/3 OTE O:1.12/7 EOR
%   B3:0/9  ILCB_LED_ON  "Turns on the instrument latch control box lights when at the zenith." %
%   I:1.18/3  SAD_LATCH2_CLS  "Saddle latch 2 closed status." %
%   O:1.12/7  SAD_LATCH2_CLS_LED  "ILCB Saddle latch 2 closed status LED" %
% Rung: 54 %
SOR XIC B3:0/9 XIC I:1.17/12 OTE O:1.13/9 EOR
%   B3:0/9  ILCB_LED_ON  "Turns on the instrument latch control box lights when at the zenith." %
%   I:1.17/12  SAFETY_LATCH1_OPN  "Protection bolt 1 open status." %
%   O:1.13/9  SAF_LATCH1_OPN_LED  "ILCB Protection bolt 1 open LED" %

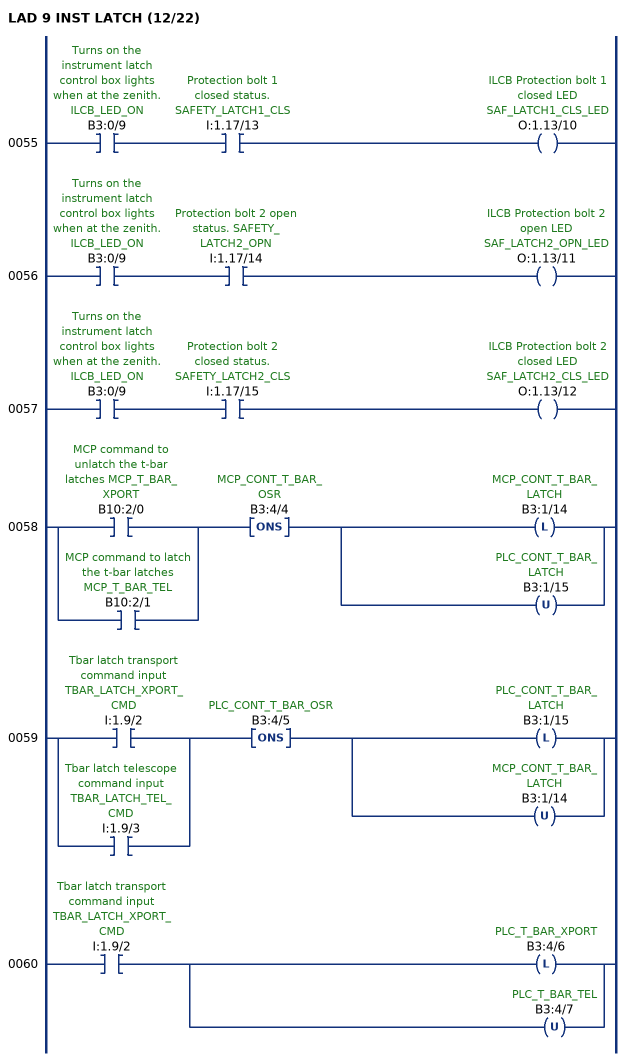
% Rung: 55 %
SOR XIC B3:0/9 XIC I:1.17/13 OTE O:1.13/10 EOR
%   B3:0/9  ILCB_LED_ON  "Turns on the instrument latch control box lights when at the zenith." %
%   I:1.17/13  SAFETY_LATCH1_CLS  "Protection bolt 1 closed status." %
%   O:1.13/10  SAF_LATCH1_CLS_LED  "ILCB Protection bolt 1 closed LED" %
% Rung: 56 %
SOR XIC B3:0/9 XIC I:1.17/14 OTE O:1.13/11 EOR
%   B3:0/9  ILCB_LED_ON  "Turns on the instrument latch control box lights when at the zenith." %
%   I:1.17/14  SAFETY_LATCH2_OPN  "Protection bolt 2 open status." %
%   O:1.13/11  SAF_LATCH2_OPN_LED  "ILCB Protection bolt 2 open LED" %
% Rung: 57 %
SOR XIC B3:0/9 XIC I:1.17/15 OTE O:1.13/12 EOR
%   B3:0/9  ILCB_LED_ON  "Turns on the instrument latch control box lights when at the zenith." %
%   I:1.17/15  SAFETY_LATCH2_CLS  "Protection bolt 2 closed status." %
%   O:1.13/12  SAF_LATCH2_CLS_LED  "ILCB Protection bolt 2 closed LED" %
% Rung: 58 %
SOR BST XIC B10:2/0 NXB XIC B10:2/1 BND OSR B3:4/4 BST OTL B3:1/14 NXB OTU B3:1/15 BND EOR
%   B10:2/0  MCP_T_BAR_XPORT  "MCP command to unlatch the t-bar latches" %
%   B10:2/1  MCP_T_BAR_TEL  "MCP command to latch the t-bar latches" %
%   B3:4/4  MCP_CONT_T_BAR_OSR %
%   B3:1/14  MCP_CONT_T_BAR_LATCH %
%   B3:1/15  PLC_CONT_T_BAR_LATCH %
% Rung: 59 %
SOR BST XIC I:1.9/2 NXB XIC I:1.9/3 BND OSR B3:4/5 BST OTL B3:1/15 NXB OTU B3:1/14 BND EOR
%   I:1.9/2  TBAR_LATCH_XPORT_CMD  "Tbar latch transport command input" %
%   I:1.9/3  TBAR_LATCH_TEL_CMD  "Tbar latch telescope command input" %
%   B3:4/5  PLC_CONT_T_BAR_OSR %
%   B3:1/15  PLC_CONT_T_BAR_LATCH %
%   B3:1/14  MCP_CONT_T_BAR_LATCH %
% Rung: 60 %
SOR XIC I:1.9/2 BST OTL B3:4/6 NXB OTU B3:4/7 BND EOR
%   I:1.9/2  TBAR_LATCH_XPORT_CMD  "Tbar latch transport command input" %
%   B3:4/6  PLC_T_BAR_XPORT %
%   B3:4/7  PLC_T_BAR_TEL %

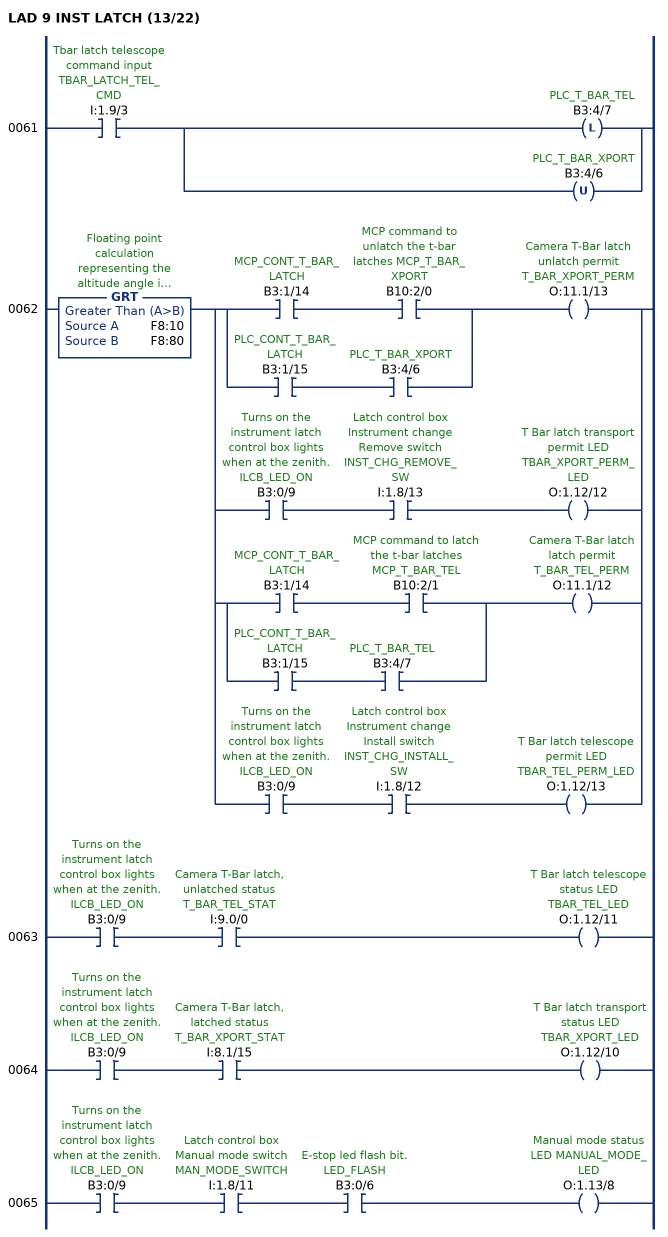
% Rung: 61 %
SOR XIC I:1.9/3 BST OTL B3:4/7 NXB OTU B3:4/6 BND EOR
%   I:1.9/3  TBAR_LATCH_TEL_CMD  "Tbar latch telescope command input" %
%   B3:4/7  PLC_T_BAR_TEL %
%   B3:4/6  PLC_T_BAR_XPORT %
% Rung: 62 %
SOR GRT F8:10 F8:80 BST BST BST XIC B3:1/14 XIC B10:2/0 NXB XIC B3:1/15 XIC B3:4/6 BND OTE O:11.1/13 NXB XIC B3:0/9 XIC I:1.8/13 OTE O:1.12/12 BND NXB BST BST XIC B3:1/14 XIC B10:2/1 NXB XIC B3:1/15 XIC B3:4/7 BND OTE O:11.1/12 NXB XIC B3:0/9 XIC I:1.8/12 OTE O:1.12/13 BND BND EOR
%   F8:10  ALT_ANGLE  "Floating point calculation representing the altitude angle in degrees." %
%   F8:80  INST_CHG_LOW_LMT  "The Lower altitude limit to allow instrument change operations" %
%   B3:1/14  MCP_CONT_T_BAR_LATCH %
%   B10:2/0  MCP_T_BAR_XPORT  "MCP command to unlatch the t-bar latches" %
%   B3:1/15  PLC_CONT_T_BAR_LATCH %
%   B3:4/6  PLC_T_BAR_XPORT %
%   O:11.1/13  T_BAR_XPORT_PERM  "Camera T-Bar latch unlatch permit" %
%   B3:0/9  ILCB_LED_ON  "Turns on the instrument latch control box lights when at the zenith." %
%   I:1.8/13  INST_CHG_REMOVE_SW  "Latch control box Instrument change Remove switch" %
%   O:1.12/12  TBAR_XPORT_PERM_LED  "T Bar latch transport permit LED" %
%   B10:2/1  MCP_T_BAR_TEL  "MCP command to latch the t-bar latches" %
%   B3:4/7  PLC_T_BAR_TEL %
%   O:11.1/12  T_BAR_TEL_PERM  "Camera T-Bar latch latch permit" %
%   I:1.8/12  INST_CHG_INSTALL_SW  "Latch control box Instrument change Install switch" %
%   O:1.12/13  TBAR_TEL_PERM_LED  "T Bar latch telescope permit LED" %
% Rung: 63 %
SOR XIC B3:0/9 XIC I:9.0/0 OTE O:1.12/11 EOR
%   B3:0/9  ILCB_LED_ON  "Turns on the instrument latch control box lights when at the zenith." %
%   I:9.0/0  T_BAR_TEL_STAT  "Camera T-Bar latch, unlatched status" %
%   O:1.12/11  TBAR_TEL_LED  "T Bar latch telescope status LED" %
% Rung: 64 %
SOR XIC B3:0/9 XIC I:8.1/15 OTE O:1.12/10 EOR
%   B3:0/9  ILCB_LED_ON  "Turns on the instrument latch control box lights when at the zenith." %
%   I:8.1/15  T_BAR_XPORT_STAT  "Camera T-Bar latch, latched status" %
%   O:1.12/10  TBAR_XPORT_LED  "T Bar latch transport status LED" %
% Rung: 65 %
SOR XIC B3:0/9 XIC I:1.8/11 XIC B3:0/6 OTE O:1.13/8 EOR
%   B3:0/9  ILCB_LED_ON  "Turns on the instrument latch control box lights when at the zenith." %
%   I:1.8/11  MAN_MODE_SWITCH  "Latch control box Manual mode switch" %
%   B3:0/6  LED_FLASH  "E-stop led flash bit." %
%   O:1.13/8  MANUAL_MODE_LED  "Manual mode status LED" %

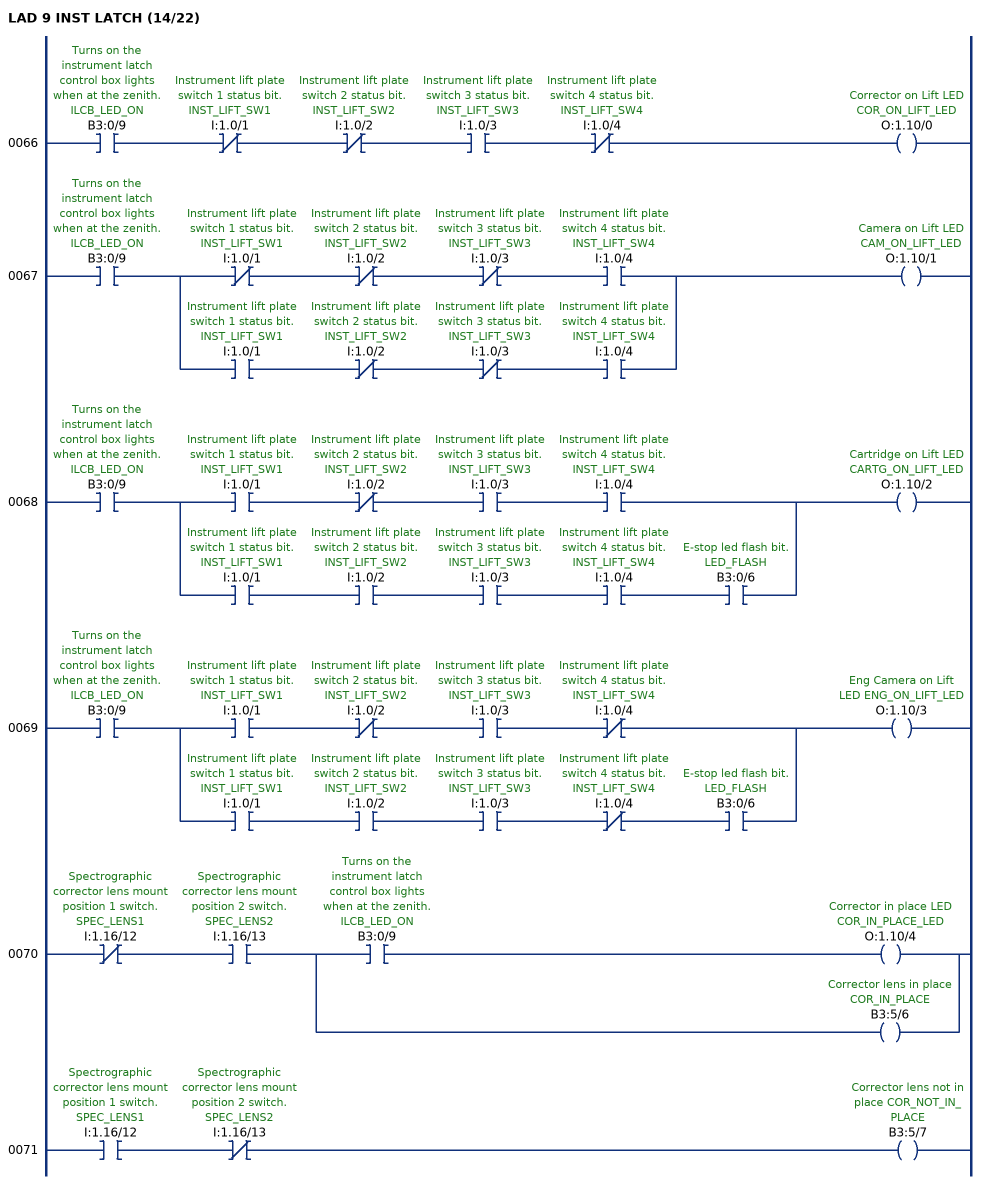
% Rung: 66 %
SOR XIC B3:0/9 XIO I:1.0/1 XIO I:1.0/2 XIC I:1.0/3 XIO I:1.0/4 OTE O:1.10/0 EOR
%   B3:0/9  ILCB_LED_ON  "Turns on the instrument latch control box lights when at the zenith." %
%   I:1.0/1  INST_LIFT_SW1  "Instrument lift plate switch 1 status bit." %
%   I:1.0/2  INST_LIFT_SW2  "Instrument lift plate switch 2 status bit." %
%   I:1.0/3  INST_LIFT_SW3  "Instrument lift plate switch 3 status bit." %
%   I:1.0/4  INST_LIFT_SW4  "Instrument lift plate switch 4 status bit." %
%   O:1.10/0  COR_ON_LIFT_LED  "Corrector on Lift LED" %
% Rung: 67 %
SOR XIC B3:0/9 BST XIO I:1.0/1 XIO I:1.0/2 XIO I:1.0/3 XIC I:1.0/4 NXB XIC I:1.0/1 XIO I:1.0/2 XIO I:1.0/3 XIC I:1.0/4 BND OTE O:1.10/1 EOR
%   B3:0/9  ILCB_LED_ON  "Turns on the instrument latch control box lights when at the zenith." %
%   I:1.0/1  INST_LIFT_SW1  "Instrument lift plate switch 1 status bit." %
%   I:1.0/2  INST_LIFT_SW2  "Instrument lift plate switch 2 status bit." %
%   I:1.0/3  INST_LIFT_SW3  "Instrument lift plate switch 3 status bit." %
%   I:1.0/4  INST_LIFT_SW4  "Instrument lift plate switch 4 status bit." %
%   O:1.10/1  CAM_ON_LIFT_LED  "Camera on Lift LED" %
% Rung: 68 %
SOR XIC B3:0/9 BST XIC I:1.0/1 XIO I:1.0/2 XIC I:1.0/3 XIC I:1.0/4 NXB XIC I:1.0/1 XIC I:1.0/2 XIC I:1.0/3 XIC I:1.0/4 XIC B3:0/6 BND OTE O:1.10/2 EOR
%   B3:0/9  ILCB_LED_ON  "Turns on the instrument latch control box lights when at the zenith." %
%   I:1.0/1  INST_LIFT_SW1  "Instrument lift plate switch 1 status bit." %
%   I:1.0/2  INST_LIFT_SW2  "Instrument lift plate switch 2 status bit." %
%   I:1.0/3  INST_LIFT_SW3  "Instrument lift plate switch 3 status bit." %
%   I:1.0/4  INST_LIFT_SW4  "Instrument lift plate switch 4 status bit." %
%   B3:0/6  LED_FLASH  "E-stop led flash bit." %
%   O:1.10/2  CARTG_ON_LIFT_LED  "Cartridge on Lift LED" %
% Rung: 69 %
SOR XIC B3:0/9 BST XIC I:1.0/1 XIO I:1.0/2 XIC I:1.0/3 XIO I:1.0/4 NXB XIC I:1.0/1 XIC I:1.0/2 XIC I:1.0/3 XIO I:1.0/4 XIC B3:0/6 BND OTE O:1.10/3 EOR
%   B3:0/9  ILCB_LED_ON  "Turns on the instrument latch control box lights when at the zenith." %
%   I:1.0/1  INST_LIFT_SW1  "Instrument lift plate switch 1 status bit." %
%   I:1.0/2  INST_LIFT_SW2  "Instrument lift plate switch 2 status bit." %
%   I:1.0/3  INST_LIFT_SW3  "Instrument lift plate switch 3 status bit." %
%   I:1.0/4  INST_LIFT_SW4  "Instrument lift plate switch 4 status bit." %
%   B3:0/6  LED_FLASH  "E-stop led flash bit." %
%   O:1.10/3  ENG_ON_LIFT_LED  "Eng Camera on Lift LED" %
% Rung: 70 %
SOR XIO I:1.16/12 XIC I:1.16/13 BST XIC B3:0/9 OTE O:1.10/4 NXB OTE B3:5/6 BND EOR
%   I:1.16/12  SPEC_LENS1  "Spectrographic corrector lens mount position 1 switch." %
%   I:1.16/13  SPEC_LENS2  "Spectrographic corrector lens mount position 2 switch." %
%   B3:0/9  ILCB_LED_ON  "Turns on the instrument latch control box lights when at the zenith." %
%   O:1.10/4  COR_IN_PLACE_LED  "Corrector in place LED" %
%   B3:5/6  COR_IN_PLACE  "Corrector lens in place" %
% Rung: 71 %
SOR XIC I:1.16/12 XIO I:1.16/13 OTE B3:5/7 EOR
%   I:1.16/12  SPEC_LENS1  "Spectrographic corrector lens mount position 1 switch." %
%   I:1.16/13  SPEC_LENS2  "Spectrographic corrector lens mount position 2 switch." %
%   B3:5/7  COR_NOT_IN_PLACE  "Corrector lens not in place" %

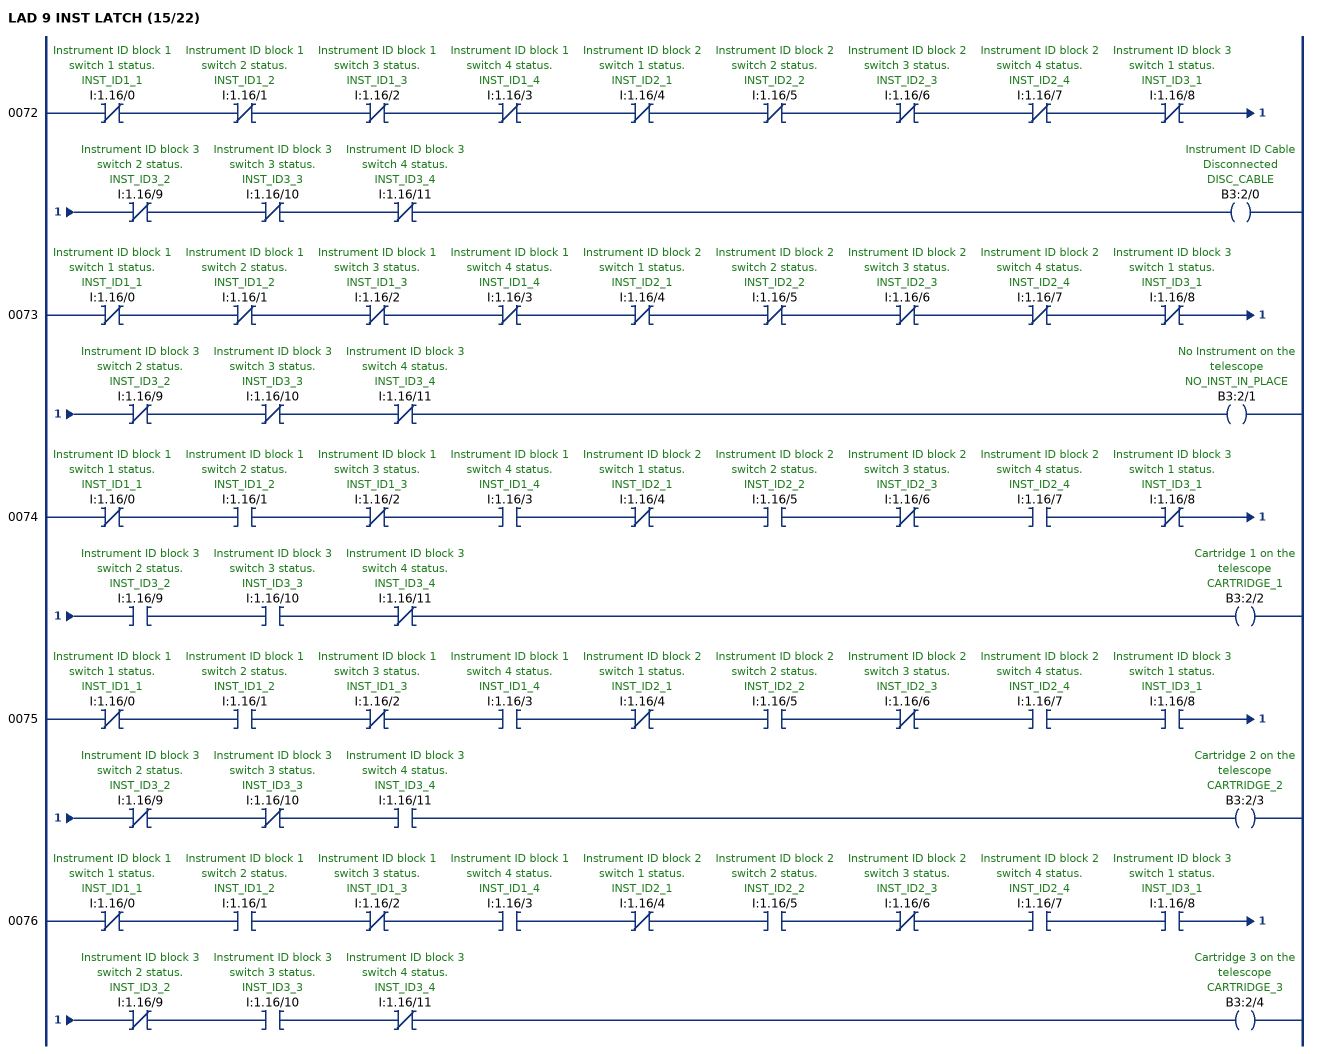
% Rung: 72 %
SOR XIO I:1.16/0 XIO I:1.16/1 XIO I:1.16/2 XIO I:1.16/3 XIO I:1.16/4 XIO I:1.16/5 XIO I:1.16/6 XIO I:1.16/7 XIO I:1.16/8 XIO I:1.16/9 XIO I:1.16/10 XIO I:1.16/11 OTE B3:2/0 EOR
%   I:1.16/0  INST_ID1_1  "Instrument ID block 1 switch 1 status." %
%   I:1.16/1  INST_ID1_2  "Instrument ID block 1 switch 2 status." %
%   I:1.16/2  INST_ID1_3  "Instrument ID block 1 switch 3 status." %
%   I:1.16/3  INST_ID1_4  "Instrument ID block 1 switch 4 status." %
%   I:1.16/4  INST_ID2_1  "Instrument ID block 2 switch 1 status." %
%   I:1.16/5  INST_ID2_2  "Instrument ID block 2 switch 2 status." %
%   I:1.16/6  INST_ID2_3  "Instrument ID block 2 switch 3 status." %
%   I:1.16/7  INST_ID2_4  "Instrument ID block 2 switch 4 status." %
%   I:1.16/8  INST_ID3_1  "Instrument ID block 3 switch 1 status." %
%   I:1.16/9  INST_ID3_2  "Instrument ID block 3 switch 2 status." %
%   I:1.16/10  INST_ID3_3  "Instrument ID block 3 switch 3 status." %
%   I:1.16/11  INST_ID3_4  "Instrument ID block 3 switch 4 status." %
%   B3:2/0  DISC_CABLE  "Instrument ID Cable Disconnected" %
% Rung: 73 %
SOR XIO I:1.16/0 XIO I:1.16/1 XIO I:1.16/2 XIO I:1.16/3 XIO I:1.16/4 XIO I:1.16/5 XIO I:1.16/6 XIO I:1.16/7 XIO I:1.16/8 XIO I:1.16/9 XIO I:1.16/10 XIO I:1.16/11 OTE B3:2/1 EOR
%   I:1.16/0  INST_ID1_1  "Instrument ID block 1 switch 1 status." %
%   I:1.16/1  INST_ID1_2  "Instrument ID block 1 switch 2 status." %
%   I:1.16/2  INST_ID1_3  "Instrument ID block 1 switch 3 status." %
%   I:1.16/3  INST_ID1_4  "Instrument ID block 1 switch 4 status." %
%   I:1.16/4  INST_ID2_1  "Instrument ID block 2 switch 1 status." %
%   I:1.16/5  INST_ID2_2  "Instrument ID block 2 switch 2 status." %
%   I:1.16/6  INST_ID2_3  "Instrument ID block 2 switch 3 status." %
%   I:1.16/7  INST_ID2_4  "Instrument ID block 2 switch 4 status." %
%   I:1.16/8  INST_ID3_1  "Instrument ID block 3 switch 1 status." %
%   I:1.16/9  INST_ID3_2  "Instrument ID block 3 switch 2 status." %
%   I:1.16/10  INST_ID3_3  "Instrument ID block 3 switch 3 status." %
%   I:1.16/11  INST_ID3_4  "Instrument ID block 3 switch 4 status." %
%   B3:2/1  NO_INST_IN_PLACE  "No Instrument on the telescope" %
% Rung: 74 %
SOR XIO I:1.16/0 XIC I:1.16/1 XIO I:1.16/2 XIC I:1.16/3 XIO I:1.16/4 XIC I:1.16/5 XIO I:1.16/6 XIC I:1.16/7 XIO I:1.16/8 XIC I:1.16/9 XIC I:1.16/10 XIO I:1.16/11 OTE B3:2/2 EOR
%   I:1.16/0  INST_ID1_1  "Instrument ID block 1 switch 1 status." %
%   I:1.16/1  INST_ID1_2  "Instrument ID block 1 switch 2 status." %
%   I:1.16/2  INST_ID1_3  "Instrument ID block 1 switch 3 status." %
%   I:1.16/3  INST_ID1_4  "Instrument ID block 1 switch 4 status." %
%   I:1.16/4  INST_ID2_1  "Instrument ID block 2 switch 1 status." %
%   I:1.16/5  INST_ID2_2  "Instrument ID block 2 switch 2 status." %
%   I:1.16/6  INST_ID2_3  "Instrument ID block 2 switch 3 status." %
%   I:1.16/7  INST_ID2_4  "Instrument ID block 2 switch 4 status." %
%   I:1.16/8  INST_ID3_1  "Instrument ID block 3 switch 1 status." %
%   I:1.16/9  INST_ID3_2  "Instrument ID block 3 switch 2 status." %
%   I:1.16/10  INST_ID3_3  "Instrument ID block 3 switch 3 status." %
%   I:1.16/11  INST_ID3_4  "Instrument ID block 3 switch 4 status." %
%   B3:2/2  CARTRIDGE_1  "Cartridge 1 on the telescope" %
% Rung: 75 %
SOR XIO I:1.16/0 XIC I:1.16/1 XIO I:1.16/2 XIC I:1.16/3 XIO I:1.16/4 XIC I:1.16/5 XIO I:1.16/6 XIC I:1.16/7 XIC I:1.16/8 XIO I:1.16/9 XIO I:1.16/10 XIC I:1.16/11 OTE B3:2/3 EOR
%   I:1.16/0  INST_ID1_1  "Instrument ID block 1 switch 1 status." %
%   I:1.16/1  INST_ID1_2  "Instrument ID block 1 switch 2 status." %
%   I:1.16/2  INST_ID1_3  "Instrument ID block 1 switch 3 status." %
%   I:1.16/3  INST_ID1_4  "Instrument ID block 1 switch 4 status." %
%   I:1.16/4  INST_ID2_1  "Instrument ID block 2 switch 1 status." %
%   I:1.16/5  INST_ID2_2  "Instrument ID block 2 switch 2 status." %
%   I:1.16/6  INST_ID2_3  "Instrument ID block 2 switch 3 status." %
%   I:1.16/7  INST_ID2_4  "Instrument ID block 2 switch 4 status." %
%   I:1.16/8  INST_ID3_1  "Instrument ID block 3 switch 1 status." %
%   I:1.16/9  INST_ID3_2  "Instrument ID block 3 switch 2 status." %
%   I:1.16/10  INST_ID3_3  "Instrument ID block 3 switch 3 status." %
%   I:1.16/11  INST_ID3_4  "Instrument ID block 3 switch 4 status." %
%   B3:2/3  CARTRIDGE_2  "Cartridge 2 on the telescope" %
% Rung: 76 %
SOR XIO I:1.16/0 XIC I:1.16/1 XIO I:1.16/2 XIC I:1.16/3 XIO I:1.16/4 XIC I:1.16/5 XIO I:1.16/6 XIC I:1.16/7 XIC I:1.16/8 XIO I:1.16/9 XIC I:1.16/10 XIO I:1.16/11 OTE B3:2/4 EOR
%   I:1.16/0  INST_ID1_1  "Instrument ID block 1 switch 1 status." %
%   I:1.16/1  INST_ID1_2  "Instrument ID block 1 switch 2 status." %
%   I:1.16/2  INST_ID1_3  "Instrument ID block 1 switch 3 status." %
%   I:1.16/3  INST_ID1_4  "Instrument ID block 1 switch 4 status." %
%   I:1.16/4  INST_ID2_1  "Instrument ID block 2 switch 1 status." %
%   I:1.16/5  INST_ID2_2  "Instrument ID block 2 switch 2 status." %
%   I:1.16/6  INST_ID2_3  "Instrument ID block 2 switch 3 status." %
%   I:1.16/7  INST_ID2_4  "Instrument ID block 2 switch 4 status." %
%   I:1.16/8  INST_ID3_1  "Instrument ID block 3 switch 1 status." %
%   I:1.16/9  INST_ID3_2  "Instrument ID block 3 switch 2 status." %
%   I:1.16/10  INST_ID3_3  "Instrument ID block 3 switch 3 status." %
%   I:1.16/11  INST_ID3_4  "Instrument ID block 3 switch 4 status." %
%   B3:2/4  CARTRIDGE_3  "Cartridge 3 on the telescope" %

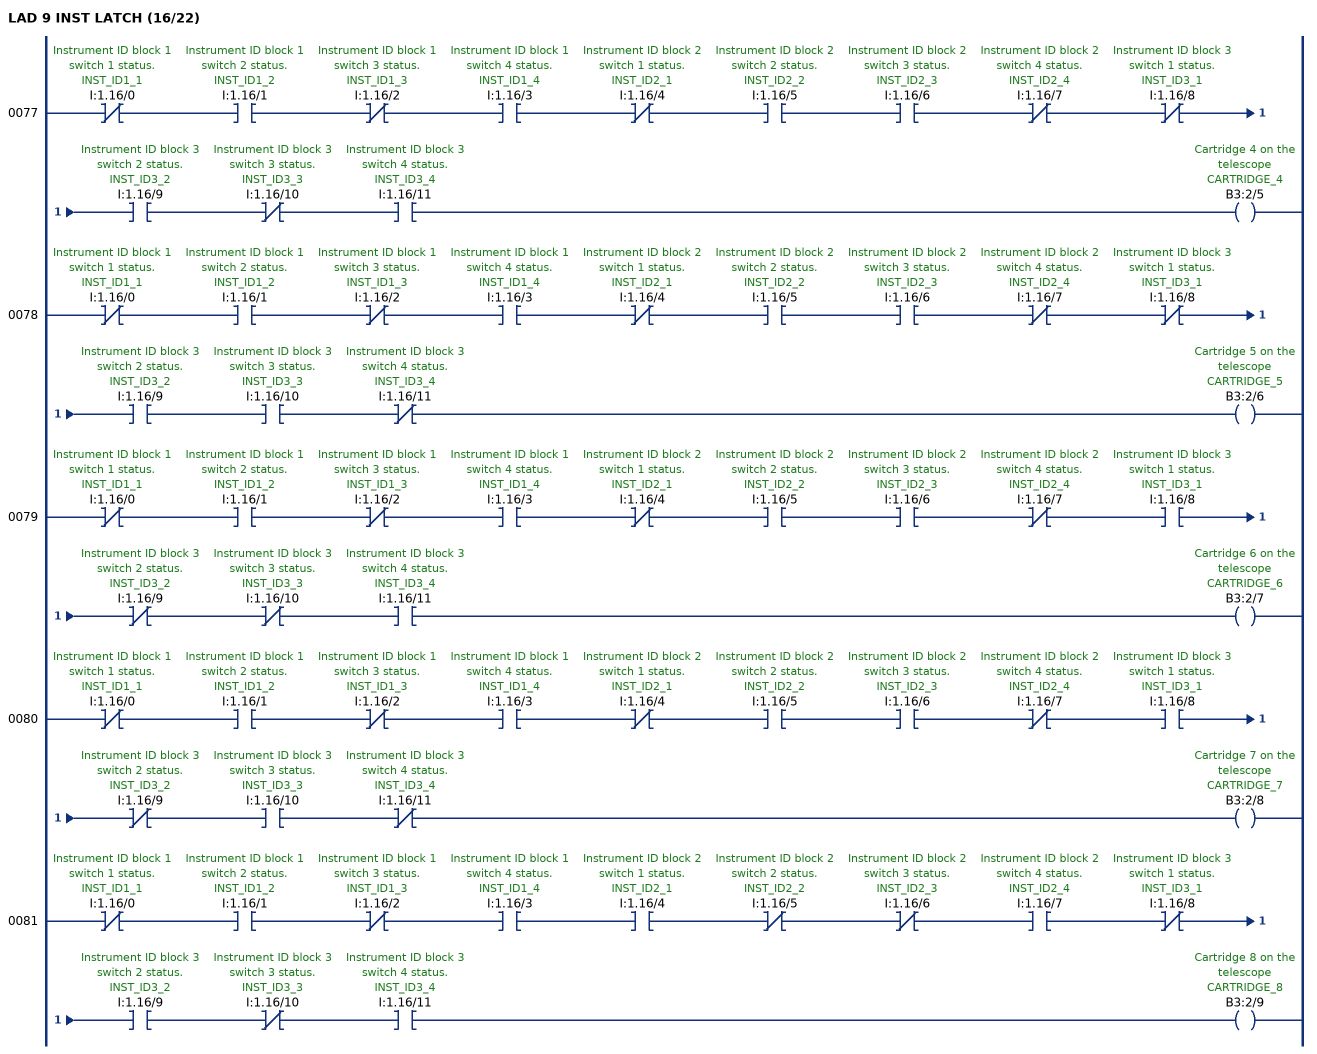
% Rung: 77 %
SOR XIO I:1.16/0 XIC I:1.16/1 XIO I:1.16/2 XIC I:1.16/3 XIO I:1.16/4 XIC I:1.16/5 XIC I:1.16/6 XIO I:1.16/7 XIO I:1.16/8 XIC I:1.16/9 XIO I:1.16/10 XIC I:1.16/11 OTE B3:2/5 EOR
%   I:1.16/0  INST_ID1_1  "Instrument ID block 1 switch 1 status." %
%   I:1.16/1  INST_ID1_2  "Instrument ID block 1 switch 2 status." %
%   I:1.16/2  INST_ID1_3  "Instrument ID block 1 switch 3 status." %
%   I:1.16/3  INST_ID1_4  "Instrument ID block 1 switch 4 status." %
%   I:1.16/4  INST_ID2_1  "Instrument ID block 2 switch 1 status." %
%   I:1.16/5  INST_ID2_2  "Instrument ID block 2 switch 2 status." %
%   I:1.16/6  INST_ID2_3  "Instrument ID block 2 switch 3 status." %
%   I:1.16/7  INST_ID2_4  "Instrument ID block 2 switch 4 status." %
%   I:1.16/8  INST_ID3_1  "Instrument ID block 3 switch 1 status." %
%   I:1.16/9  INST_ID3_2  "Instrument ID block 3 switch 2 status." %
%   I:1.16/10  INST_ID3_3  "Instrument ID block 3 switch 3 status." %
%   I:1.16/11  INST_ID3_4  "Instrument ID block 3 switch 4 status." %
%   B3:2/5  CARTRIDGE_4  "Cartridge 4 on the telescope" %
% Rung: 78 %
SOR XIO I:1.16/0 XIC I:1.16/1 XIO I:1.16/2 XIC I:1.16/3 XIO I:1.16/4 XIC I:1.16/5 XIC I:1.16/6 XIO I:1.16/7 XIO I:1.16/8 XIC I:1.16/9 XIC I:1.16/10 XIO I:1.16/11 OTE B3:2/6 EOR
%   I:1.16/0  INST_ID1_1  "Instrument ID block 1 switch 1 status." %
%   I:1.16/1  INST_ID1_2  "Instrument ID block 1 switch 2 status." %
%   I:1.16/2  INST_ID1_3  "Instrument ID block 1 switch 3 status." %
%   I:1.16/3  INST_ID1_4  "Instrument ID block 1 switch 4 status." %
%   I:1.16/4  INST_ID2_1  "Instrument ID block 2 switch 1 status." %
%   I:1.16/5  INST_ID2_2  "Instrument ID block 2 switch 2 status." %
%   I:1.16/6  INST_ID2_3  "Instrument ID block 2 switch 3 status." %
%   I:1.16/7  INST_ID2_4  "Instrument ID block 2 switch 4 status." %
%   I:1.16/8  INST_ID3_1  "Instrument ID block 3 switch 1 status." %
%   I:1.16/9  INST_ID3_2  "Instrument ID block 3 switch 2 status." %
%   I:1.16/10  INST_ID3_3  "Instrument ID block 3 switch 3 status." %
%   I:1.16/11  INST_ID3_4  "Instrument ID block 3 switch 4 status." %
%   B3:2/6  CARTRIDGE_5  "Cartridge 5 on the telescope" %
% Rung: 79 %
SOR XIO I:1.16/0 XIC I:1.16/1 XIO I:1.16/2 XIC I:1.16/3 XIO I:1.16/4 XIC I:1.16/5 XIC I:1.16/6 XIO I:1.16/7 XIC I:1.16/8 XIO I:1.16/9 XIO I:1.16/10 XIC I:1.16/11 OTE B3:2/7 EOR
%   I:1.16/0  INST_ID1_1  "Instrument ID block 1 switch 1 status." %
%   I:1.16/1  INST_ID1_2  "Instrument ID block 1 switch 2 status." %
%   I:1.16/2  INST_ID1_3  "Instrument ID block 1 switch 3 status." %
%   I:1.16/3  INST_ID1_4  "Instrument ID block 1 switch 4 status." %
%   I:1.16/4  INST_ID2_1  "Instrument ID block 2 switch 1 status." %
%   I:1.16/5  INST_ID2_2  "Instrument ID block 2 switch 2 status." %
%   I:1.16/6  INST_ID2_3  "Instrument ID block 2 switch 3 status." %
%   I:1.16/7  INST_ID2_4  "Instrument ID block 2 switch 4 status." %
%   I:1.16/8  INST_ID3_1  "Instrument ID block 3 switch 1 status." %
%   I:1.16/9  INST_ID3_2  "Instrument ID block 3 switch 2 status." %
%   I:1.16/10  INST_ID3_3  "Instrument ID block 3 switch 3 status." %
%   I:1.16/11  INST_ID3_4  "Instrument ID block 3 switch 4 status." %
%   B3:2/7  CARTRIDGE_6  "Cartridge 6 on the telescope" %
% Rung: 80 %
SOR XIO I:1.16/0 XIC I:1.16/1 XIO I:1.16/2 XIC I:1.16/3 XIO I:1.16/4 XIC I:1.16/5 XIC I:1.16/6 XIO I:1.16/7 XIC I:1.16/8 XIO I:1.16/9 XIC I:1.16/10 XIO I:1.16/11 OTE B3:2/8 EOR
%   I:1.16/0  INST_ID1_1  "Instrument ID block 1 switch 1 status." %
%   I:1.16/1  INST_ID1_2  "Instrument ID block 1 switch 2 status." %
%   I:1.16/2  INST_ID1_3  "Instrument ID block 1 switch 3 status." %
%   I:1.16/3  INST_ID1_4  "Instrument ID block 1 switch 4 status." %
%   I:1.16/4  INST_ID2_1  "Instrument ID block 2 switch 1 status." %
%   I:1.16/5  INST_ID2_2  "Instrument ID block 2 switch 2 status." %
%   I:1.16/6  INST_ID2_3  "Instrument ID block 2 switch 3 status." %
%   I:1.16/7  INST_ID2_4  "Instrument ID block 2 switch 4 status." %
%   I:1.16/8  INST_ID3_1  "Instrument ID block 3 switch 1 status." %
%   I:1.16/9  INST_ID3_2  "Instrument ID block 3 switch 2 status." %
%   I:1.16/10  INST_ID3_3  "Instrument ID block 3 switch 3 status." %
%   I:1.16/11  INST_ID3_4  "Instrument ID block 3 switch 4 status." %
%   B3:2/8  CARTRIDGE_7  "Cartridge 7 on the telescope" %
% Rung: 81 %
SOR XIO I:1.16/0 XIC I:1.16/1 XIO I:1.16/2 XIC I:1.16/3 XIC I:1.16/4 XIO I:1.16/5 XIO I:1.16/6 XIC I:1.16/7 XIO I:1.16/8 XIC I:1.16/9 XIO I:1.16/10 XIC I:1.16/11 OTE B3:2/9 EOR
%   I:1.16/0  INST_ID1_1  "Instrument ID block 1 switch 1 status." %
%   I:1.16/1  INST_ID1_2  "Instrument ID block 1 switch 2 status." %
%   I:1.16/2  INST_ID1_3  "Instrument ID block 1 switch 3 status." %
%   I:1.16/3  INST_ID1_4  "Instrument ID block 1 switch 4 status." %
%   I:1.16/4  INST_ID2_1  "Instrument ID block 2 switch 1 status." %
%   I:1.16/5  INST_ID2_2  "Instrument ID block 2 switch 2 status." %
%   I:1.16/6  INST_ID2_3  "Instrument ID block 2 switch 3 status." %
%   I:1.16/7  INST_ID2_4  "Instrument ID block 2 switch 4 status." %
%   I:1.16/8  INST_ID3_1  "Instrument ID block 3 switch 1 status." %
%   I:1.16/9  INST_ID3_2  "Instrument ID block 3 switch 2 status." %
%   I:1.16/10  INST_ID3_3  "Instrument ID block 3 switch 3 status." %
%   I:1.16/11  INST_ID3_4  "Instrument ID block 3 switch 4 status." %
%   B3:2/9  CARTRIDGE_8  "Cartridge 8 on the telescope" %

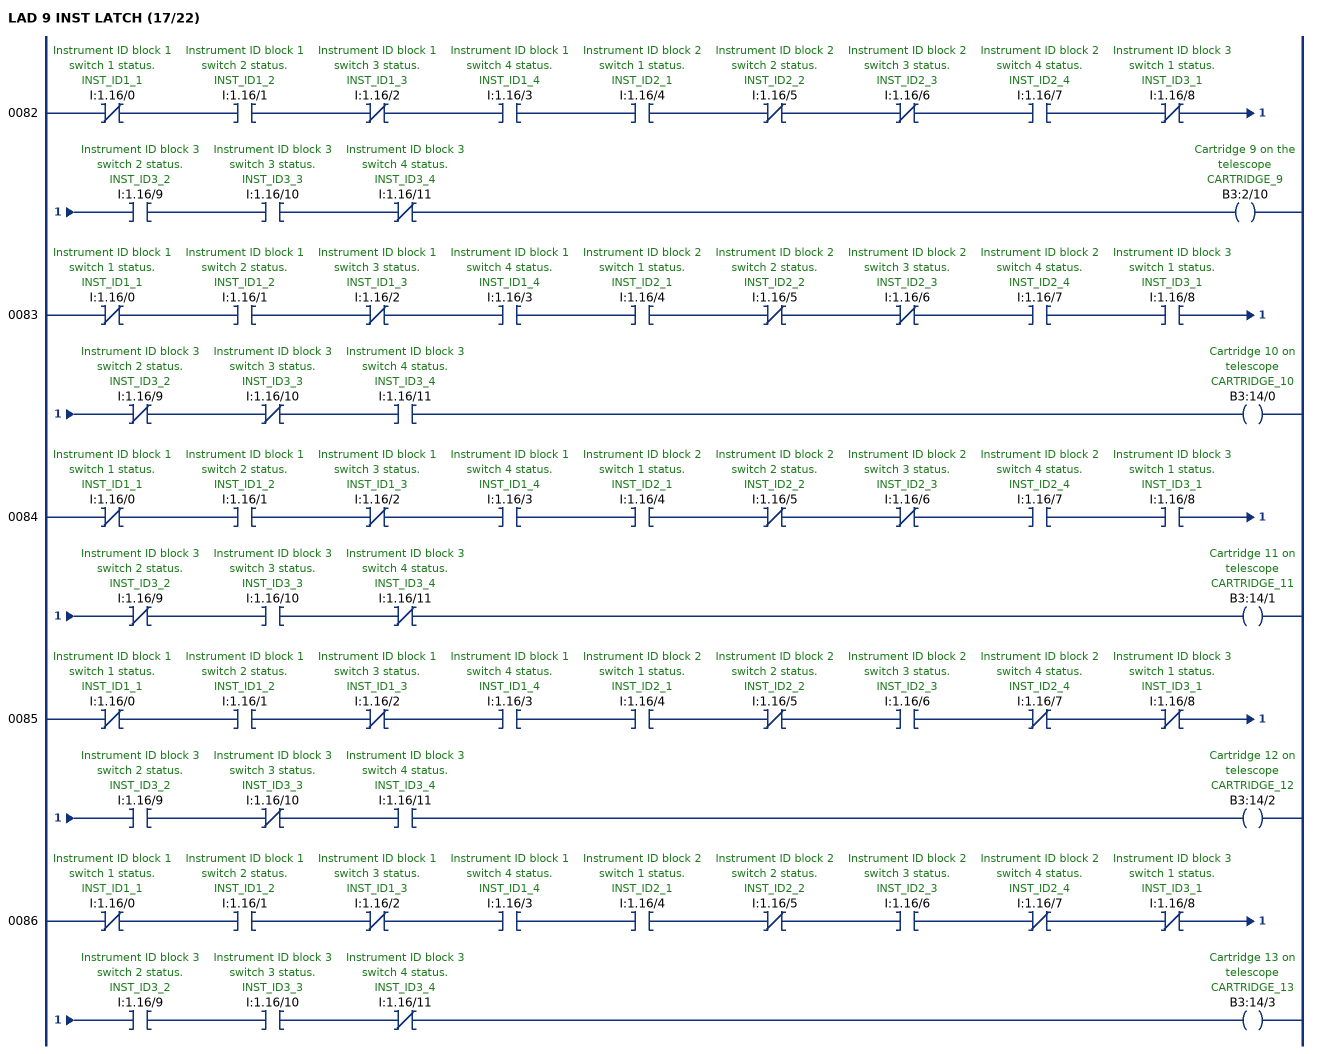
% Rung: 82 %
SOR XIO I:1.16/0 XIC I:1.16/1 XIO I:1.16/2 XIC I:1.16/3 XIC I:1.16/4 XIO I:1.16/5 XIO I:1.16/6 XIC I:1.16/7 XIO I:1.16/8 XIC I:1.16/9 XIC I:1.16/10 XIO I:1.16/11 OTE B3:2/10 EOR
%   I:1.16/0  INST_ID1_1  "Instrument ID block 1 switch 1 status." %
%   I:1.16/1  INST_ID1_2  "Instrument ID block 1 switch 2 status." %
%   I:1.16/2  INST_ID1_3  "Instrument ID block 1 switch 3 status." %
%   I:1.16/3  INST_ID1_4  "Instrument ID block 1 switch 4 status." %
%   I:1.16/4  INST_ID2_1  "Instrument ID block 2 switch 1 status." %
%   I:1.16/5  INST_ID2_2  "Instrument ID block 2 switch 2 status." %
%   I:1.16/6  INST_ID2_3  "Instrument ID block 2 switch 3 status." %
%   I:1.16/7  INST_ID2_4  "Instrument ID block 2 switch 4 status." %
%   I:1.16/8  INST_ID3_1  "Instrument ID block 3 switch 1 status." %
%   I:1.16/9  INST_ID3_2  "Instrument ID block 3 switch 2 status." %
%   I:1.16/10  INST_ID3_3  "Instrument ID block 3 switch 3 status." %
%   I:1.16/11  INST_ID3_4  "Instrument ID block 3 switch 4 status." %
%   B3:2/10  CARTRIDGE_9  "Cartridge 9 on the telescope" %
% Rung: 83 %
SOR XIO I:1.16/0 XIC I:1.16/1 XIO I:1.16/2 XIC I:1.16/3 XIC I:1.16/4 XIO I:1.16/5 XIO I:1.16/6 XIC I:1.16/7 XIC I:1.16/8 XIO I:1.16/9 XIO I:1.16/10 XIC I:1.16/11 OTE B3:14/0 EOR
%   I:1.16/0  INST_ID1_1  "Instrument ID block 1 switch 1 status." %
%   I:1.16/1  INST_ID1_2  "Instrument ID block 1 switch 2 status." %
%   I:1.16/2  INST_ID1_3  "Instrument ID block 1 switch 3 status." %
%   I:1.16/3  INST_ID1_4  "Instrument ID block 1 switch 4 status." %
%   I:1.16/4  INST_ID2_1  "Instrument ID block 2 switch 1 status." %
%   I:1.16/5  INST_ID2_2  "Instrument ID block 2 switch 2 status." %
%   I:1.16/6  INST_ID2_3  "Instrument ID block 2 switch 3 status." %
%   I:1.16/7  INST_ID2_4  "Instrument ID block 2 switch 4 status." %
%   I:1.16/8  INST_ID3_1  "Instrument ID block 3 switch 1 status." %
%   I:1.16/9  INST_ID3_2  "Instrument ID block 3 switch 2 status." %
%   I:1.16/10  INST_ID3_3  "Instrument ID block 3 switch 3 status." %
%   I:1.16/11  INST_ID3_4  "Instrument ID block 3 switch 4 status." %
%   B3:14/0  CARTRIDGE_10  "Cartridge 10 on telescope" %
% Rung: 84 %
SOR XIO I:1.16/0 XIC I:1.16/1 XIO I:1.16/2 XIC I:1.16/3 XIC I:1.16/4 XIO I:1.16/5 XIO I:1.16/6 XIC I:1.16/7 XIC I:1.16/8 XIO I:1.16/9 XIC I:1.16/10 XIO I:1.16/11 OTE B3:14/1 EOR
%   I:1.16/0  INST_ID1_1  "Instrument ID block 1 switch 1 status." %
%   I:1.16/1  INST_ID1_2  "Instrument ID block 1 switch 2 status." %
%   I:1.16/2  INST_ID1_3  "Instrument ID block 1 switch 3 status." %
%   I:1.16/3  INST_ID1_4  "Instrument ID block 1 switch 4 status." %
%   I:1.16/4  INST_ID2_1  "Instrument ID block 2 switch 1 status." %
%   I:1.16/5  INST_ID2_2  "Instrument ID block 2 switch 2 status." %
%   I:1.16/6  INST_ID2_3  "Instrument ID block 2 switch 3 status." %
%   I:1.16/7  INST_ID2_4  "Instrument ID block 2 switch 4 status." %
%   I:1.16/8  INST_ID3_1  "Instrument ID block 3 switch 1 status." %
%   I:1.16/9  INST_ID3_2  "Instrument ID block 3 switch 2 status." %
%   I:1.16/10  INST_ID3_3  "Instrument ID block 3 switch 3 status." %
%   I:1.16/11  INST_ID3_4  "Instrument ID block 3 switch 4 status." %
%   B3:14/1  CARTRIDGE_11  "Cartridge 11 on telescope" %
% Rung: 85 %
SOR XIO I:1.16/0 XIC I:1.16/1 XIO I:1.16/2 XIC I:1.16/3 XIC I:1.16/4 XIO I:1.16/5 XIC I:1.16/6 XIO I:1.16/7 XIO I:1.16/8 XIC I:1.16/9 XIO I:1.16/10 XIC I:1.16/11 OTE B3:14/2 EOR
%   I:1.16/0  INST_ID1_1  "Instrument ID block 1 switch 1 status." %
%   I:1.16/1  INST_ID1_2  "Instrument ID block 1 switch 2 status." %
%   I:1.16/2  INST_ID1_3  "Instrument ID block 1 switch 3 status." %
%   I:1.16/3  INST_ID1_4  "Instrument ID block 1 switch 4 status." %
%   I:1.16/4  INST_ID2_1  "Instrument ID block 2 switch 1 status." %
%   I:1.16/5  INST_ID2_2  "Instrument ID block 2 switch 2 status." %
%   I:1.16/6  INST_ID2_3  "Instrument ID block 2 switch 3 status." %
%   I:1.16/7  INST_ID2_4  "Instrument ID block 2 switch 4 status." %
%   I:1.16/8  INST_ID3_1  "Instrument ID block 3 switch 1 status." %
%   I:1.16/9  INST_ID3_2  "Instrument ID block 3 switch 2 status." %
%   I:1.16/10  INST_ID3_3  "Instrument ID block 3 switch 3 status." %
%   I:1.16/11  INST_ID3_4  "Instrument ID block 3 switch 4 status." %
%   B3:14/2  CARTRIDGE_12  "Cartridge 12 on telescope" %
% Rung: 86 %
SOR XIO I:1.16/0 XIC I:1.16/1 XIO I:1.16/2 XIC I:1.16/3 XIC I:1.16/4 XIO I:1.16/5 XIC I:1.16/6 XIO I:1.16/7 XIO I:1.16/8 XIC I:1.16/9 XIC I:1.16/10 XIO I:1.16/11 OTE B3:14/3 EOR
%   I:1.16/0  INST_ID1_1  "Instrument ID block 1 switch 1 status." %
%   I:1.16/1  INST_ID1_2  "Instrument ID block 1 switch 2 status." %
%   I:1.16/2  INST_ID1_3  "Instrument ID block 1 switch 3 status." %
%   I:1.16/3  INST_ID1_4  "Instrument ID block 1 switch 4 status." %
%   I:1.16/4  INST_ID2_1  "Instrument ID block 2 switch 1 status." %
%   I:1.16/5  INST_ID2_2  "Instrument ID block 2 switch 2 status." %
%   I:1.16/6  INST_ID2_3  "Instrument ID block 2 switch 3 status." %
%   I:1.16/7  INST_ID2_4  "Instrument ID block 2 switch 4 status." %
%   I:1.16/8  INST_ID3_1  "Instrument ID block 3 switch 1 status." %
%   I:1.16/9  INST_ID3_2  "Instrument ID block 3 switch 2 status." %
%   I:1.16/10  INST_ID3_3  "Instrument ID block 3 switch 3 status." %
%   I:1.16/11  INST_ID3_4  "Instrument ID block 3 switch 4 status." %
%   B3:14/3  CARTRIDGE_13  "Cartridge 13 on telescope" %

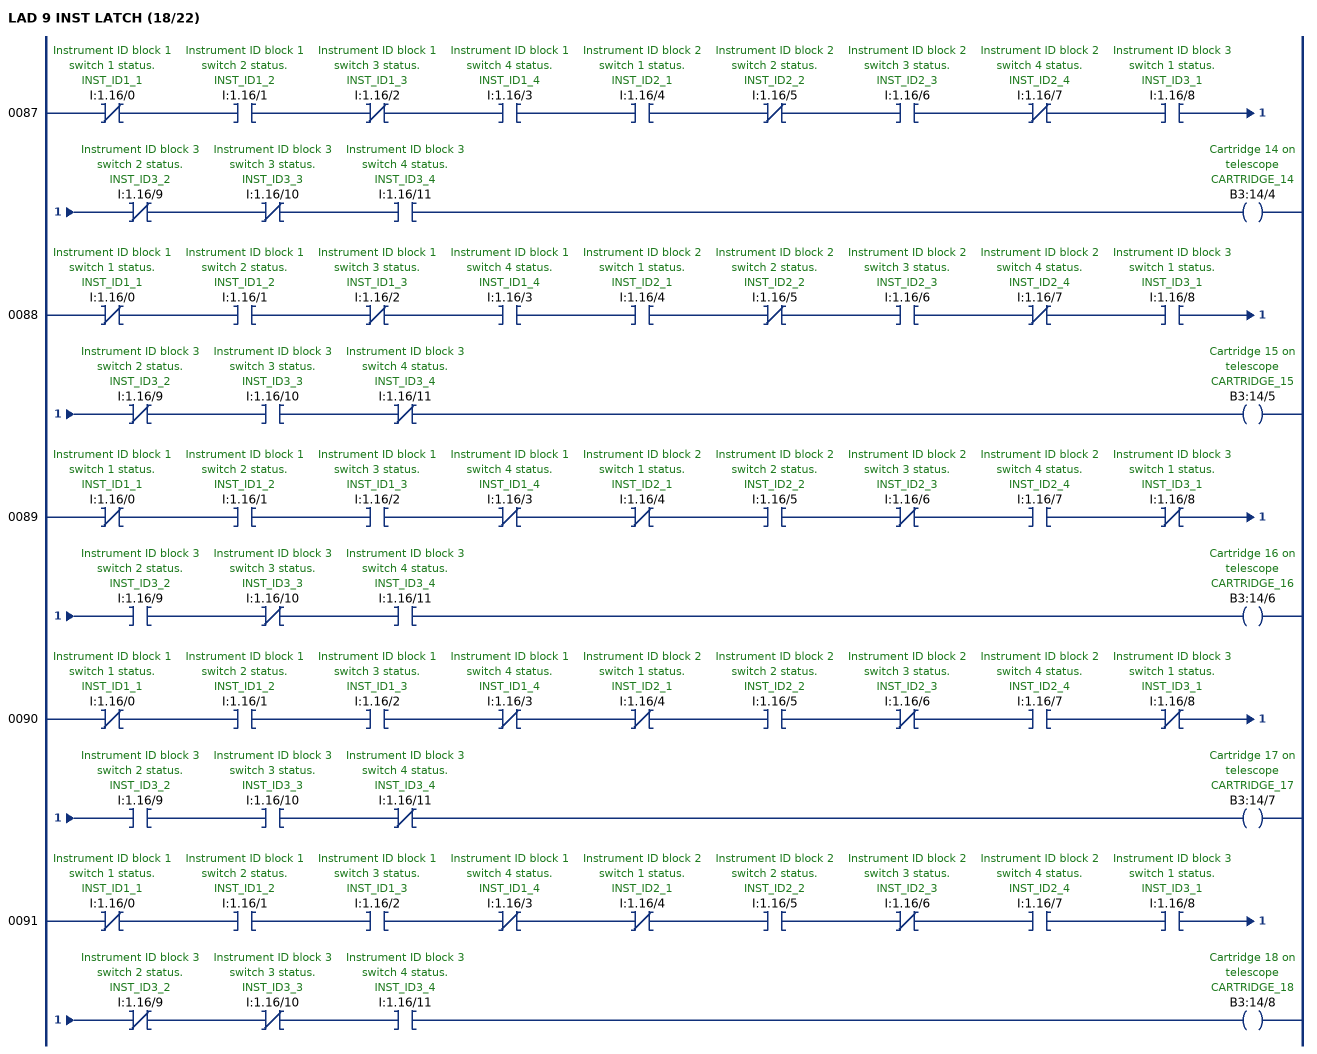
% Rung: 87 %
SOR XIO I:1.16/0 XIC I:1.16/1 XIO I:1.16/2 XIC I:1.16/3 XIC I:1.16/4 XIO I:1.16/5 XIC I:1.16/6 XIO I:1.16/7 XIC I:1.16/8 XIO I:1.16/9 XIO I:1.16/10 XIC I:1.16/11 OTE B3:14/4 EOR
%   I:1.16/0  INST_ID1_1  "Instrument ID block 1 switch 1 status." %
%   I:1.16/1  INST_ID1_2  "Instrument ID block 1 switch 2 status." %
%   I:1.16/2  INST_ID1_3  "Instrument ID block 1 switch 3 status." %
%   I:1.16/3  INST_ID1_4  "Instrument ID block 1 switch 4 status." %
%   I:1.16/4  INST_ID2_1  "Instrument ID block 2 switch 1 status." %
%   I:1.16/5  INST_ID2_2  "Instrument ID block 2 switch 2 status." %
%   I:1.16/6  INST_ID2_3  "Instrument ID block 2 switch 3 status." %
%   I:1.16/7  INST_ID2_4  "Instrument ID block 2 switch 4 status." %
%   I:1.16/8  INST_ID3_1  "Instrument ID block 3 switch 1 status." %
%   I:1.16/9  INST_ID3_2  "Instrument ID block 3 switch 2 status." %
%   I:1.16/10  INST_ID3_3  "Instrument ID block 3 switch 3 status." %
%   I:1.16/11  INST_ID3_4  "Instrument ID block 3 switch 4 status." %
%   B3:14/4  CARTRIDGE_14  "Cartridge 14 on telescope" %
% Rung: 88 %
SOR XIO I:1.16/0 XIC I:1.16/1 XIO I:1.16/2 XIC I:1.16/3 XIC I:1.16/4 XIO I:1.16/5 XIC I:1.16/6 XIO I:1.16/7 XIC I:1.16/8 XIO I:1.16/9 XIC I:1.16/10 XIO I:1.16/11 OTE B3:14/5 EOR
%   I:1.16/0  INST_ID1_1  "Instrument ID block 1 switch 1 status." %
%   I:1.16/1  INST_ID1_2  "Instrument ID block 1 switch 2 status." %
%   I:1.16/2  INST_ID1_3  "Instrument ID block 1 switch 3 status." %
%   I:1.16/3  INST_ID1_4  "Instrument ID block 1 switch 4 status." %
%   I:1.16/4  INST_ID2_1  "Instrument ID block 2 switch 1 status." %
%   I:1.16/5  INST_ID2_2  "Instrument ID block 2 switch 2 status." %
%   I:1.16/6  INST_ID2_3  "Instrument ID block 2 switch 3 status." %
%   I:1.16/7  INST_ID2_4  "Instrument ID block 2 switch 4 status." %
%   I:1.16/8  INST_ID3_1  "Instrument ID block 3 switch 1 status." %
%   I:1.16/9  INST_ID3_2  "Instrument ID block 3 switch 2 status." %
%   I:1.16/10  INST_ID3_3  "Instrument ID block 3 switch 3 status." %
%   I:1.16/11  INST_ID3_4  "Instrument ID block 3 switch 4 status." %
%   B3:14/5  CARTRIDGE_15  "Cartridge 15 on telescope" %
% Rung: 89 %
SOR XIO I:1.16/0 XIC I:1.16/1 XIC I:1.16/2 XIO I:1.16/3 XIO I:1.16/4 XIC I:1.16/5 XIO I:1.16/6 XIC I:1.16/7 XIO I:1.16/8 XIC I:1.16/9 XIO I:1.16/10 XIC I:1.16/11 OTE B3:14/6 EOR
%   I:1.16/0  INST_ID1_1  "Instrument ID block 1 switch 1 status." %
%   I:1.16/1  INST_ID1_2  "Instrument ID block 1 switch 2 status." %
%   I:1.16/2  INST_ID1_3  "Instrument ID block 1 switch 3 status." %
%   I:1.16/3  INST_ID1_4  "Instrument ID block 1 switch 4 status." %
%   I:1.16/4  INST_ID2_1  "Instrument ID block 2 switch 1 status." %
%   I:1.16/5  INST_ID2_2  "Instrument ID block 2 switch 2 status." %
%   I:1.16/6  INST_ID2_3  "Instrument ID block 2 switch 3 status." %
%   I:1.16/7  INST_ID2_4  "Instrument ID block 2 switch 4 status." %
%   I:1.16/8  INST_ID3_1  "Instrument ID block 3 switch 1 status." %
%   I:1.16/9  INST_ID3_2  "Instrument ID block 3 switch 2 status." %
%   I:1.16/10  INST_ID3_3  "Instrument ID block 3 switch 3 status." %
%   I:1.16/11  INST_ID3_4  "Instrument ID block 3 switch 4 status." %
%   B3:14/6  CARTRIDGE_16  "Cartridge 16 on telescope" %
% Rung: 90 %
SOR XIO I:1.16/0 XIC I:1.16/1 XIC I:1.16/2 XIO I:1.16/3 XIO I:1.16/4 XIC I:1.16/5 XIO I:1.16/6 XIC I:1.16/7 XIO I:1.16/8 XIC I:1.16/9 XIC I:1.16/10 XIO I:1.16/11 OTE B3:14/7 EOR
%   I:1.16/0  INST_ID1_1  "Instrument ID block 1 switch 1 status." %
%   I:1.16/1  INST_ID1_2  "Instrument ID block 1 switch 2 status." %
%   I:1.16/2  INST_ID1_3  "Instrument ID block 1 switch 3 status." %
%   I:1.16/3  INST_ID1_4  "Instrument ID block 1 switch 4 status." %
%   I:1.16/4  INST_ID2_1  "Instrument ID block 2 switch 1 status." %
%   I:1.16/5  INST_ID2_2  "Instrument ID block 2 switch 2 status." %
%   I:1.16/6  INST_ID2_3  "Instrument ID block 2 switch 3 status." %
%   I:1.16/7  INST_ID2_4  "Instrument ID block 2 switch 4 status." %
%   I:1.16/8  INST_ID3_1  "Instrument ID block 3 switch 1 status." %
%   I:1.16/9  INST_ID3_2  "Instrument ID block 3 switch 2 status." %
%   I:1.16/10  INST_ID3_3  "Instrument ID block 3 switch 3 status." %
%   I:1.16/11  INST_ID3_4  "Instrument ID block 3 switch 4 status." %
%   B3:14/7  CARTRIDGE_17  "Cartridge 17 on telescope" %
% Rung: 91 %
SOR XIO I:1.16/0 XIC I:1.16/1 XIC I:1.16/2 XIO I:1.16/3 XIO I:1.16/4 XIC I:1.16/5 XIO I:1.16/6 XIC I:1.16/7 XIC I:1.16/8 XIO I:1.16/9 XIO I:1.16/10 XIC I:1.16/11 OTE B3:14/8 EOR
%   I:1.16/0  INST_ID1_1  "Instrument ID block 1 switch 1 status." %
%   I:1.16/1  INST_ID1_2  "Instrument ID block 1 switch 2 status." %
%   I:1.16/2  INST_ID1_3  "Instrument ID block 1 switch 3 status." %
%   I:1.16/3  INST_ID1_4  "Instrument ID block 1 switch 4 status." %
%   I:1.16/4  INST_ID2_1  "Instrument ID block 2 switch 1 status." %
%   I:1.16/5  INST_ID2_2  "Instrument ID block 2 switch 2 status." %
%   I:1.16/6  INST_ID2_3  "Instrument ID block 2 switch 3 status." %
%   I:1.16/7  INST_ID2_4  "Instrument ID block 2 switch 4 status." %
%   I:1.16/8  INST_ID3_1  "Instrument ID block 3 switch 1 status." %
%   I:1.16/9  INST_ID3_2  "Instrument ID block 3 switch 2 status." %
%   I:1.16/10  INST_ID3_3  "Instrument ID block 3 switch 3 status." %
%   I:1.16/11  INST_ID3_4  "Instrument ID block 3 switch 4 status." %
%   B3:14/8  CARTRIDGE_18  "Cartridge 18 on telescope" %

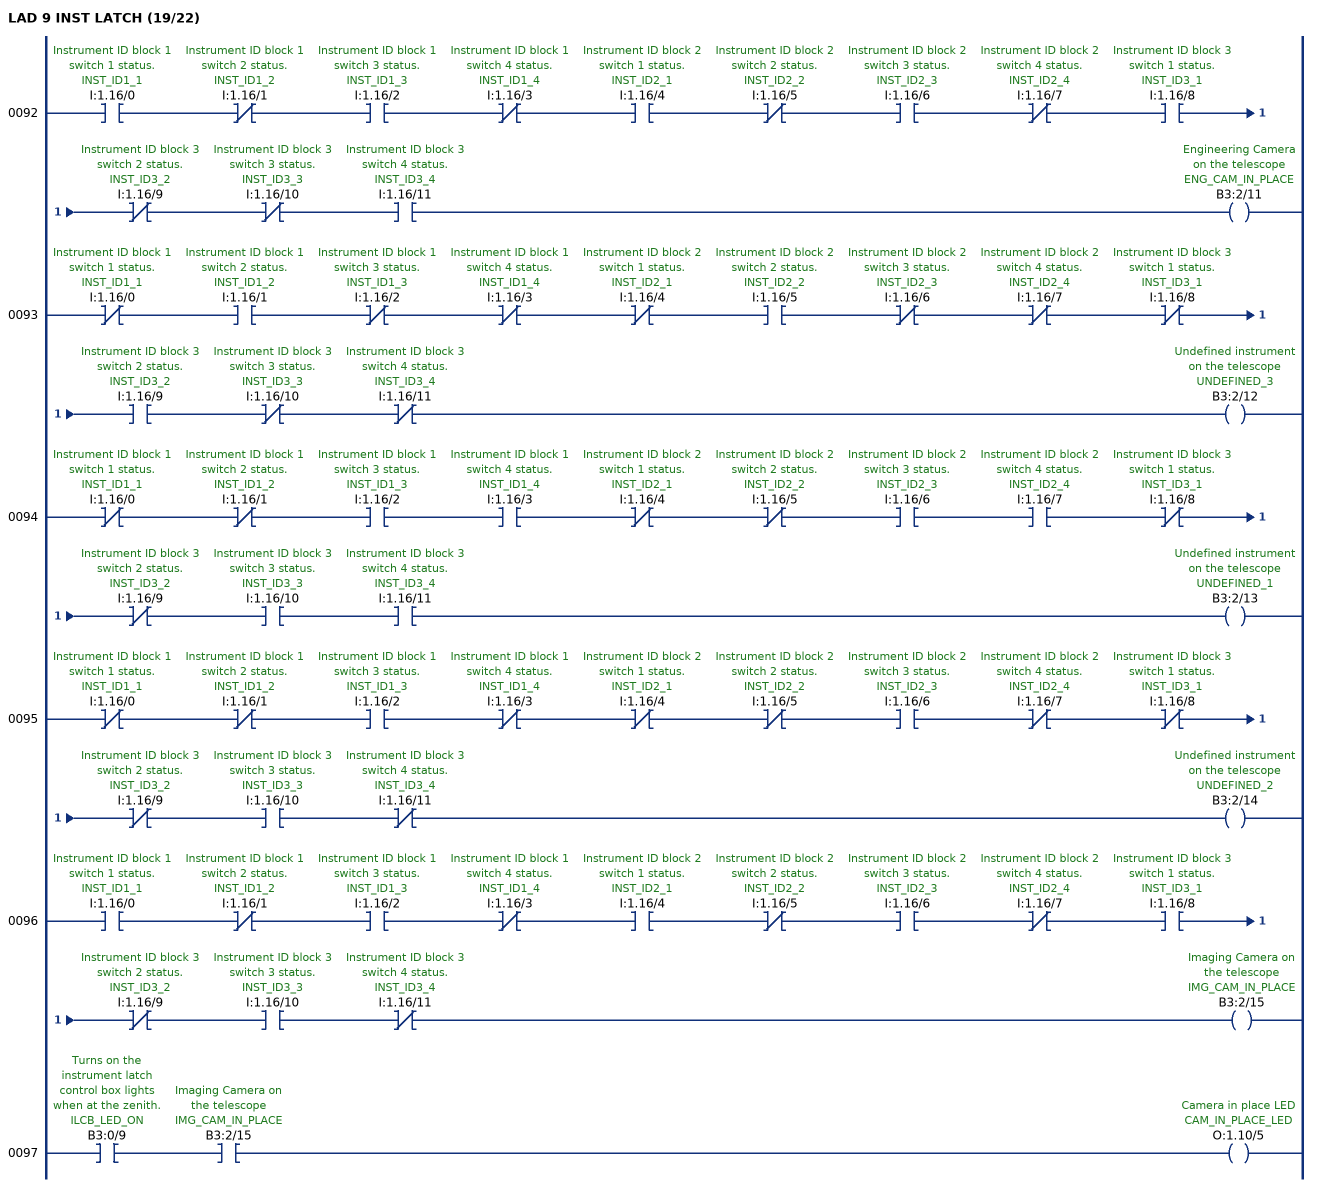
% Rung: 92 %
SOR XIC I:1.16/0 XIO I:1.16/1 XIC I:1.16/2 XIO I:1.16/3 XIC I:1.16/4 XIO I:1.16/5 XIC I:1.16/6 XIO I:1.16/7 XIC I:1.16/8 XIO I:1.16/9 XIO I:1.16/10 XIC I:1.16/11 OTE B3:2/11 EOR
%   I:1.16/0  INST_ID1_1  "Instrument ID block 1 switch 1 status." %
%   I:1.16/1  INST_ID1_2  "Instrument ID block 1 switch 2 status." %
%   I:1.16/2  INST_ID1_3  "Instrument ID block 1 switch 3 status." %
%   I:1.16/3  INST_ID1_4  "Instrument ID block 1 switch 4 status." %
%   I:1.16/4  INST_ID2_1  "Instrument ID block 2 switch 1 status." %
%   I:1.16/5  INST_ID2_2  "Instrument ID block 2 switch 2 status." %
%   I:1.16/6  INST_ID2_3  "Instrument ID block 2 switch 3 status." %
%   I:1.16/7  INST_ID2_4  "Instrument ID block 2 switch 4 status." %
%   I:1.16/8  INST_ID3_1  "Instrument ID block 3 switch 1 status." %
%   I:1.16/9  INST_ID3_2  "Instrument ID block 3 switch 2 status." %
%   I:1.16/10  INST_ID3_3  "Instrument ID block 3 switch 3 status." %
%   I:1.16/11  INST_ID3_4  "Instrument ID block 3 switch 4 status." %
%   B3:2/11  ENG_CAM_IN_PLACE  "Engineering Camera on the telescope" %
% Rung: 93 %
SOR XIO I:1.16/0 XIC I:1.16/1 XIO I:1.16/2 XIO I:1.16/3 XIO I:1.16/4 XIC I:1.16/5 XIO I:1.16/6 XIO I:1.16/7 XIO I:1.16/8 XIC I:1.16/9 XIO I:1.16/10 XIO I:1.16/11 OTE B3:2/12 EOR
%   I:1.16/0  INST_ID1_1  "Instrument ID block 1 switch 1 status." %
%   I:1.16/1  INST_ID1_2  "Instrument ID block 1 switch 2 status." %
%   I:1.16/2  INST_ID1_3  "Instrument ID block 1 switch 3 status." %
%   I:1.16/3  INST_ID1_4  "Instrument ID block 1 switch 4 status." %
%   I:1.16/4  INST_ID2_1  "Instrument ID block 2 switch 1 status." %
%   I:1.16/5  INST_ID2_2  "Instrument ID block 2 switch 2 status." %
%   I:1.16/6  INST_ID2_3  "Instrument ID block 2 switch 3 status." %
%   I:1.16/7  INST_ID2_4  "Instrument ID block 2 switch 4 status." %
%   I:1.16/8  INST_ID3_1  "Instrument ID block 3 switch 1 status." %
%   I:1.16/9  INST_ID3_2  "Instrument ID block 3 switch 2 status." %
%   I:1.16/10  INST_ID3_3  "Instrument ID block 3 switch 3 status." %
%   I:1.16/11  INST_ID3_4  "Instrument ID block 3 switch 4 status." %
%   B3:2/12  UNDEFINED_3  "Undefined instrument on the telescope" %
% Rung: 94 %
SOR XIO I:1.16/0 XIO I:1.16/1 XIC I:1.16/2 XIC I:1.16/3 XIO I:1.16/4 XIO I:1.16/5 XIC I:1.16/6 XIC I:1.16/7 XIO I:1.16/8 XIO I:1.16/9 XIC I:1.16/10 XIC I:1.16/11 OTE B3:2/13 EOR
%   I:1.16/0  INST_ID1_1  "Instrument ID block 1 switch 1 status." %
%   I:1.16/1  INST_ID1_2  "Instrument ID block 1 switch 2 status." %
%   I:1.16/2  INST_ID1_3  "Instrument ID block 1 switch 3 status." %
%   I:1.16/3  INST_ID1_4  "Instrument ID block 1 switch 4 status." %
%   I:1.16/4  INST_ID2_1  "Instrument ID block 2 switch 1 status." %
%   I:1.16/5  INST_ID2_2  "Instrument ID block 2 switch 2 status." %
%   I:1.16/6  INST_ID2_3  "Instrument ID block 2 switch 3 status." %
%   I:1.16/7  INST_ID2_4  "Instrument ID block 2 switch 4 status." %
%   I:1.16/8  INST_ID3_1  "Instrument ID block 3 switch 1 status." %
%   I:1.16/9  INST_ID3_2  "Instrument ID block 3 switch 2 status." %
%   I:1.16/10  INST_ID3_3  "Instrument ID block 3 switch 3 status." %
%   I:1.16/11  INST_ID3_4  "Instrument ID block 3 switch 4 status." %
%   B3:2/13  UNDEFINED_1  "Undefined instrument on the telescope" %
% Rung: 95 %
SOR XIO I:1.16/0 XIO I:1.16/1 XIC I:1.16/2 XIO I:1.16/3 XIO I:1.16/4 XIO I:1.16/5 XIC I:1.16/6 XIO I:1.16/7 XIO I:1.16/8 XIO I:1.16/9 XIC I:1.16/10 XIO I:1.16/11 OTE B3:2/14 EOR
%   I:1.16/0  INST_ID1_1  "Instrument ID block 1 switch 1 status." %
%   I:1.16/1  INST_ID1_2  "Instrument ID block 1 switch 2 status." %
%   I:1.16/2  INST_ID1_3  "Instrument ID block 1 switch 3 status." %
%   I:1.16/3  INST_ID1_4  "Instrument ID block 1 switch 4 status." %
%   I:1.16/4  INST_ID2_1  "Instrument ID block 2 switch 1 status." %
%   I:1.16/5  INST_ID2_2  "Instrument ID block 2 switch 2 status." %
%   I:1.16/6  INST_ID2_3  "Instrument ID block 2 switch 3 status." %
%   I:1.16/7  INST_ID2_4  "Instrument ID block 2 switch 4 status." %
%   I:1.16/8  INST_ID3_1  "Instrument ID block 3 switch 1 status." %
%   I:1.16/9  INST_ID3_2  "Instrument ID block 3 switch 2 status." %
%   I:1.16/10  INST_ID3_3  "Instrument ID block 3 switch 3 status." %
%   I:1.16/11  INST_ID3_4  "Instrument ID block 3 switch 4 status." %
%   B3:2/14  UNDEFINED_2  "Undefined instrument on the telescope" %
% Rung: 96 %
SOR XIC I:1.16/0 XIO I:1.16/1 XIC I:1.16/2 XIO I:1.16/3 XIC I:1.16/4 XIO I:1.16/5 XIC I:1.16/6 XIO I:1.16/7 XIC I:1.16/8 XIO I:1.16/9 XIC I:1.16/10 XIO I:1.16/11 OTE B3:2/15 EOR
%   I:1.16/0  INST_ID1_1  "Instrument ID block 1 switch 1 status." %
%   I:1.16/1  INST_ID1_2  "Instrument ID block 1 switch 2 status." %
%   I:1.16/2  INST_ID1_3  "Instrument ID block 1 switch 3 status." %
%   I:1.16/3  INST_ID1_4  "Instrument ID block 1 switch 4 status." %
%   I:1.16/4  INST_ID2_1  "Instrument ID block 2 switch 1 status." %
%   I:1.16/5  INST_ID2_2  "Instrument ID block 2 switch 2 status." %
%   I:1.16/6  INST_ID2_3  "Instrument ID block 2 switch 3 status." %
%   I:1.16/7  INST_ID2_4  "Instrument ID block 2 switch 4 status." %
%   I:1.16/8  INST_ID3_1  "Instrument ID block 3 switch 1 status." %
%   I:1.16/9  INST_ID3_2  "Instrument ID block 3 switch 2 status." %
%   I:1.16/10  INST_ID3_3  "Instrument ID block 3 switch 3 status." %
%   I:1.16/11  INST_ID3_4  "Instrument ID block 3 switch 4 status." %
%   B3:2/15  IMG_CAM_IN_PLACE  "Imaging Camera on the telescope" %
% Rung: 97 %
SOR XIC B3:0/9 XIC B3:2/15 OTE O:1.10/5 EOR
%   B3:0/9  ILCB_LED_ON  "Turns on the instrument latch control box lights when at the zenith." %
%   B3:2/15  IMG_CAM_IN_PLACE  "Imaging Camera on the telescope" %
%   O:1.10/5  CAM_IN_PLACE_LED  "Camera in place LED" %

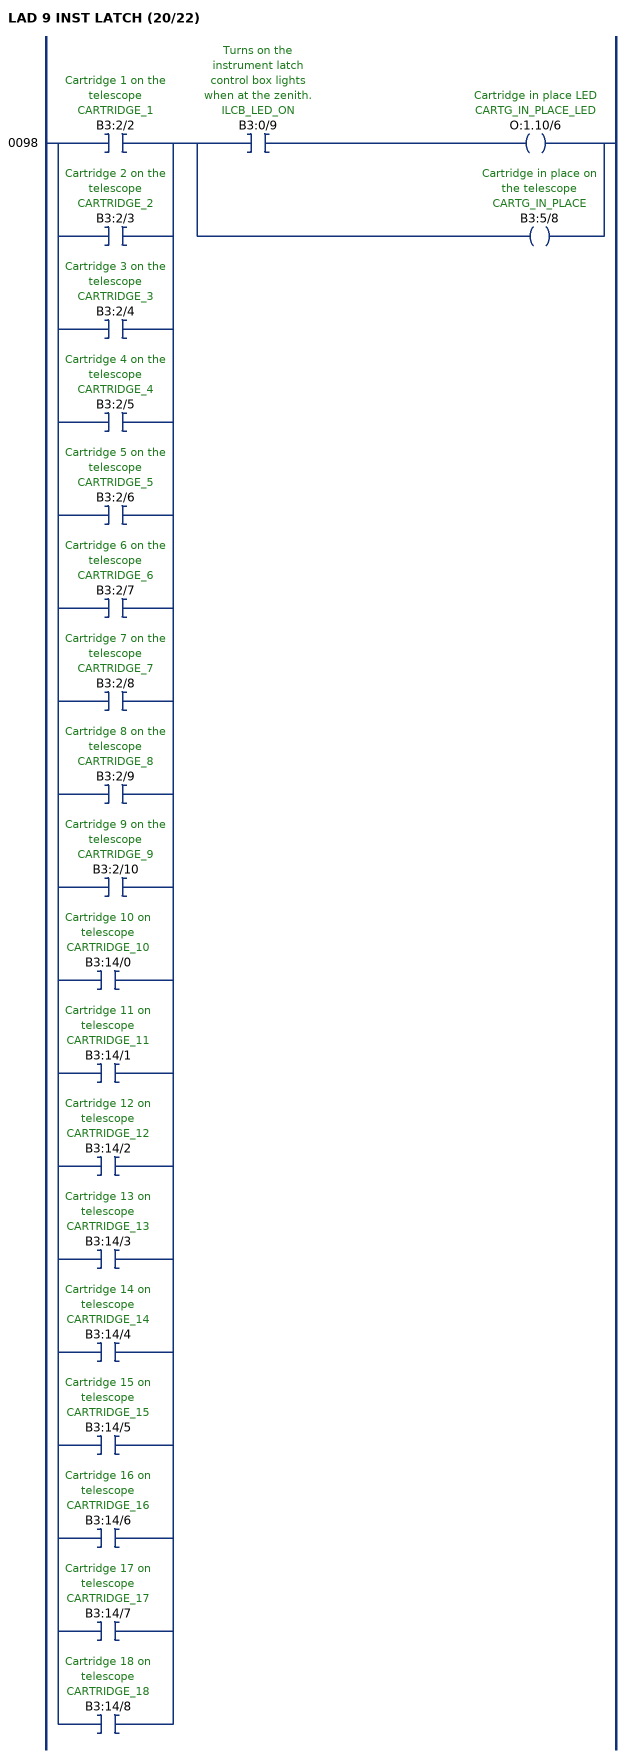
% Rung: 98 %
SOR BST XIC B3:2/2 NXB XIC B3:2/3 NXB XIC B3:2/4 NXB XIC B3:2/5 NXB XIC B3:2/6 NXB XIC B3:2/7 NXB XIC B3:2/8 NXB XIC B3:2/9 NXB XIC B3:2/10 NXB XIC B3:14/0 NXB XIC B3:14/1 NXB XIC B3:14/2 NXB XIC B3:14/3 NXB XIC B3:14/4 NXB XIC B3:14/5 NXB XIC B3:14/6 NXB BST XIC B3:14/7 NXB XIC B3:14/8 BND BND BST XIC B3:0/9 OTE O:1.10/6 NXB OTE B3:5/8 BND EOR
%   B3:2/2  CARTRIDGE_1  "Cartridge 1 on the telescope" %
%   B3:2/3  CARTRIDGE_2  "Cartridge 2 on the telescope" %
%   B3:2/4  CARTRIDGE_3  "Cartridge 3 on the telescope" %
%   B3:2/5  CARTRIDGE_4  "Cartridge 4 on the telescope" %
%   B3:2/6  CARTRIDGE_5  "Cartridge 5 on the telescope" %
%   B3:2/7  CARTRIDGE_6  "Cartridge 6 on the telescope" %
%   B3:2/8  CARTRIDGE_7  "Cartridge 7 on the telescope" %
%   B3:2/9  CARTRIDGE_8  "Cartridge 8 on the telescope" %
%   B3:2/10  CARTRIDGE_9  "Cartridge 9 on the telescope" %
%   B3:14/0  CARTRIDGE_10  "Cartridge 10 on telescope" %
%   B3:14/1  CARTRIDGE_11  "Cartridge 11 on telescope" %
%   B3:14/2  CARTRIDGE_12  "Cartridge 12 on telescope" %
%   B3:14/3  CARTRIDGE_13  "Cartridge 13 on telescope" %
%   B3:14/4  CARTRIDGE_14  "Cartridge 14 on telescope" %
%   B3:14/5  CARTRIDGE_15  "Cartridge 15 on telescope" %
%   B3:14/6  CARTRIDGE_16  "Cartridge 16 on telescope" %
%   B3:14/7  CARTRIDGE_17  "Cartridge 17 on telescope" %
%   B3:14/8  CARTRIDGE_18  "Cartridge 18 on telescope" %
%   B3:0/9  ILCB_LED_ON  "Turns on the instrument latch control box lights when at the zenith." %
%   O:1.10/6  CARTG_IN_PLACE_LED  "Cartridge in place LED" %
%   B3:5/8  CARTG_IN_PLACE  "Cartridge in place on the telescope" %

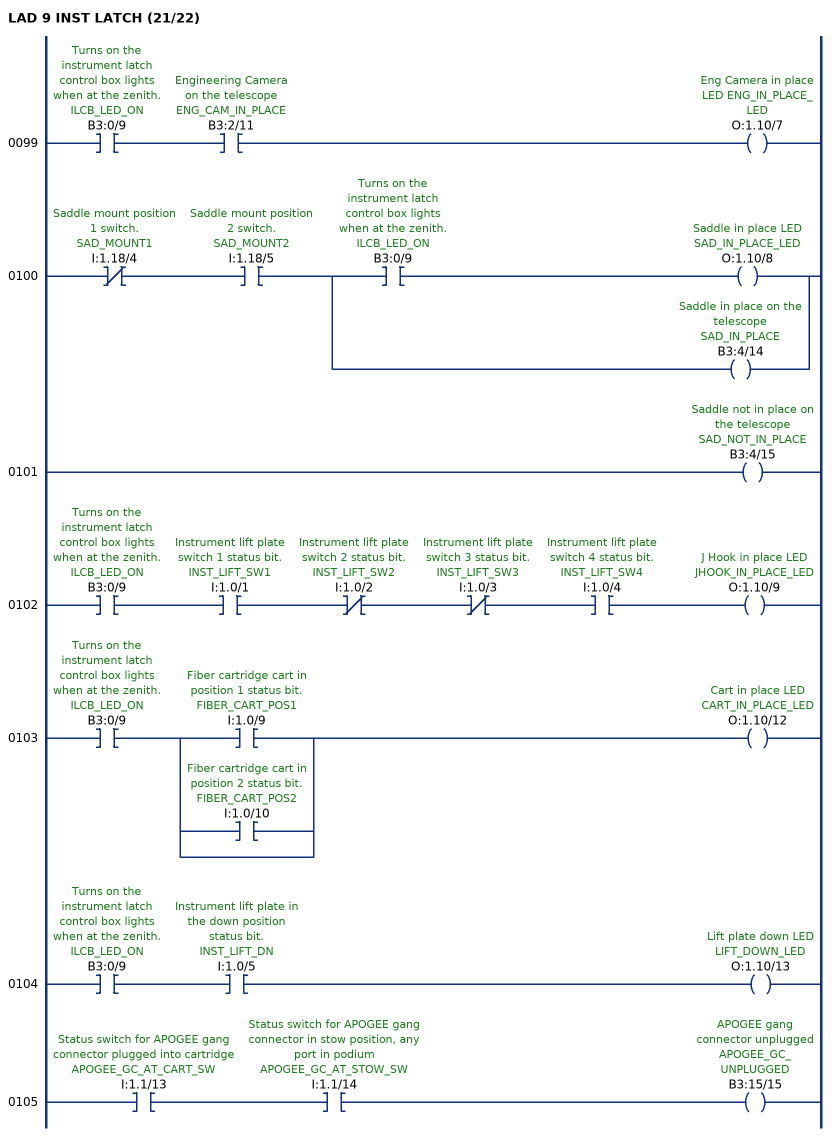
% Rung: 99 %
SOR XIC B3:0/9 XIC B3:2/11 OTE O:1.10/7 EOR
%   B3:0/9  ILCB_LED_ON  "Turns on the instrument latch control box lights when at the zenith." %
%   B3:2/11  ENG_CAM_IN_PLACE  "Engineering Camera on the telescope" %
%   O:1.10/7  ENG_IN_PLACE_LED  "Eng Camera in place LED" %
% Rung: 100 %
SOR XIO I:1.18/4 XIC I:1.18/5 BST XIC B3:0/9 OTE O:1.10/8 NXB OTE B3:4/14 BND EOR
%   I:1.18/4  SAD_MOUNT1  "Saddle mount position 1 switch." %
%   I:1.18/5  SAD_MOUNT2  "Saddle mount position 2 switch." %
%   B3:0/9  ILCB_LED_ON  "Turns on the instrument latch control box lights when at the zenith." %
%   O:1.10/8  SAD_IN_PLACE_LED  "Saddle in place LED" %
%   B3:4/14  SAD_IN_PLACE  "Saddle in place on the telescope" %
% Rung: 101 %
SOR OTE B3:4/15 EOR
%   B3:4/15  SAD_NOT_IN_PLACE  "Saddle not in place on the telescope" %
% Rung: 102 %
SOR XIC B3:0/9 XIC I:1.0/1 XIO I:1.0/2 XIO I:1.0/3 XIC I:1.0/4 OTE O:1.10/9 EOR
%   B3:0/9  ILCB_LED_ON  "Turns on the instrument latch control box lights when at the zenith." %
%   I:1.0/1  INST_LIFT_SW1  "Instrument lift plate switch 1 status bit." %
%   I:1.0/2  INST_LIFT_SW2  "Instrument lift plate switch 2 status bit." %
%   I:1.0/3  INST_LIFT_SW3  "Instrument lift plate switch 3 status bit." %
%   I:1.0/4  INST_LIFT_SW4  "Instrument lift plate switch 4 status bit." %
%   O:1.10/9  JHOOK_IN_PLACE_LED  "J Hook in place LED" %
% Rung: 103 %
SOR XIC B3:0/9 BST XIC I:1.0/9 NXB XIC I:1.0/10 NXB BND OTE O:1.10/12 EOR
%   B3:0/9  ILCB_LED_ON  "Turns on the instrument latch control box lights when at the zenith." %
%   I:1.0/9  FIBER_CART_POS1  "Fiber cartridge cart in position 1 status bit." %
%   I:1.0/10  FIBER_CART_POS2  "Fiber cartridge cart in position 2 status bit." %
%   O:1.10/12  CART_IN_PLACE_LED  "Cart in place LED" %
% Rung: 104 %
SOR XIC B3:0/9 XIC I:1.0/5 OTE O:1.10/13 EOR
%   B3:0/9  ILCB_LED_ON  "Turns on the instrument latch control box lights when at the zenith." %
%   I:1.0/5  INST_LIFT_DN  "Instrument lift plate in the down position status bit." %
%   O:1.10/13  LIFT_DOWN_LED  "Lift plate down LED" %
% Rung: 105 %
SOR XIC I:1.1/13 XIC I:1.1/14 OTE B3:15/15 EOR
%   I:1.1/13  APOGEE_GC_AT_CART_SW  "Status switch for APOGEE gang connector plugged into cartridge" %
%   I:1.1/14  APOGEE_GC_AT_STOW_SW  "Status switch for APOGEE gang connector in stow position, any port in podium" %
%   B3:15/15  APOGEE_GC_UNPLUGGED  "APOGEE gang connector unplugged" %

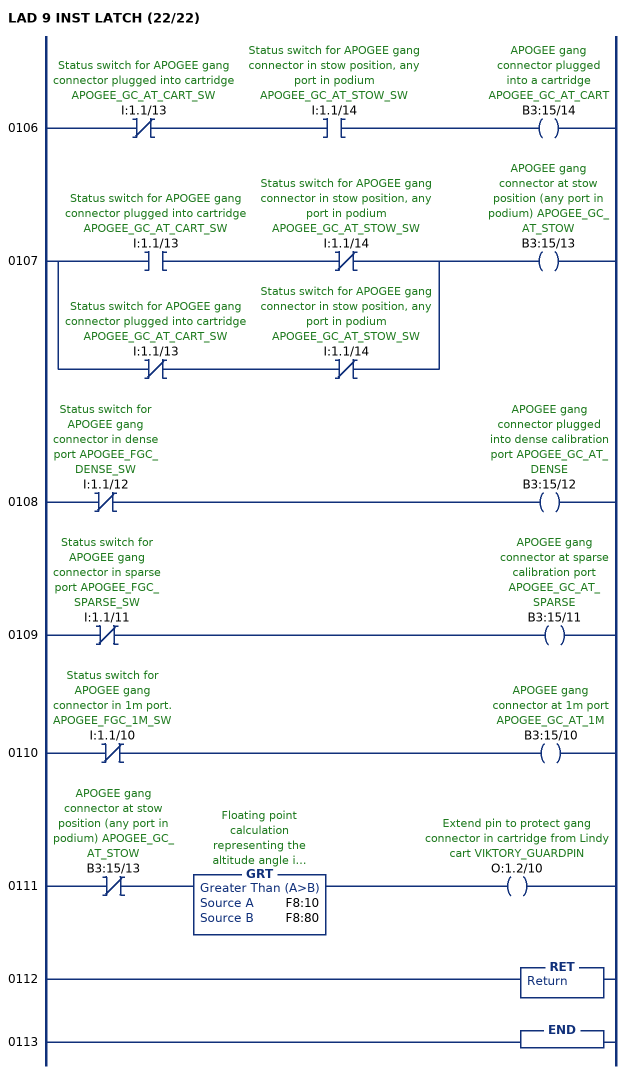
% Rung: 106 %
SOR XIO I:1.1/13 XIC I:1.1/14 OTE B3:15/14 EOR
%   I:1.1/13  APOGEE_GC_AT_CART_SW  "Status switch for APOGEE gang connector plugged into cartridge" %
%   I:1.1/14  APOGEE_GC_AT_STOW_SW  "Status switch for APOGEE gang connector in stow position, any port in podium" %
%   B3:15/14  APOGEE_GC_AT_CART  "APOGEE gang connector plugged into a cartridge" %
% Rung: 107 %
SOR BST XIC I:1.1/13 XIO I:1.1/14 NXB XIO I:1.1/13 XIO I:1.1/14 BND OTE B3:15/13 EOR
%   I:1.1/13  APOGEE_GC_AT_CART_SW  "Status switch for APOGEE gang connector plugged into cartridge" %
%   I:1.1/14  APOGEE_GC_AT_STOW_SW  "Status switch for APOGEE gang connector in stow position, any port in podium" %
%   B3:15/13  APOGEE_GC_AT_STOW  "APOGEE gang connector at stow position (any port in podium)" %
% Rung: 108 %
SOR XIO I:1.1/12 OTE B3:15/12 EOR
%   I:1.1/12  APOGEE_FGC_DENSE_SW  "Status switch for APOGEE gang connector in dense port" %
%   B3:15/12  APOGEE_GC_AT_DENSE  "APOGEE gang connector plugged into dense calibration port" %
% Rung: 109 %
SOR XIO I:1.1/11 OTE B3:15/11 EOR
%   I:1.1/11  APOGEE_FGC_SPARSE_SW  "Status switch for APOGEE gang connector in sparse port" %
%   B3:15/11  APOGEE_GC_AT_SPARSE  "APOGEE gang connector at sparse calibration port" %
% Rung: 110 %
SOR XIO I:1.1/10 OTE B3:15/10 EOR
%   I:1.1/10  APOGEE_FGC_1M_SW  "Status switch for APOGEE gang connector in 1m port." %
%   B3:15/10  APOGEE_GC_AT_1M  "APOGEE gang connector at 1m port" %
% Rung: 111 %
SOR XIO B3:15/13 GRT F8:10 F8:80 OTE O:1.2/10 EOR
%   B3:15/13  APOGEE_GC_AT_STOW  "APOGEE gang connector at stow position (any port in podium)" %
%   F8:10  ALT_ANGLE  "Floating point calculation representing the altitude angle in degrees." %
%   F8:80  INST_CHG_LOW_LMT  "The Lower altitude limit to allow instrument change operations" %
%   O:1.2/10  VIKTORY_GUARDPIN  "Extend pin to protect gang connector in cartridge from Lindy cart" %
% Rung: 112 %
SOR RET EOR
% Rung: 113 %
SOR END EOR

LADDER 10 "DATA TRANS"    % Data Transfer subroutine for DH+ link to VME %
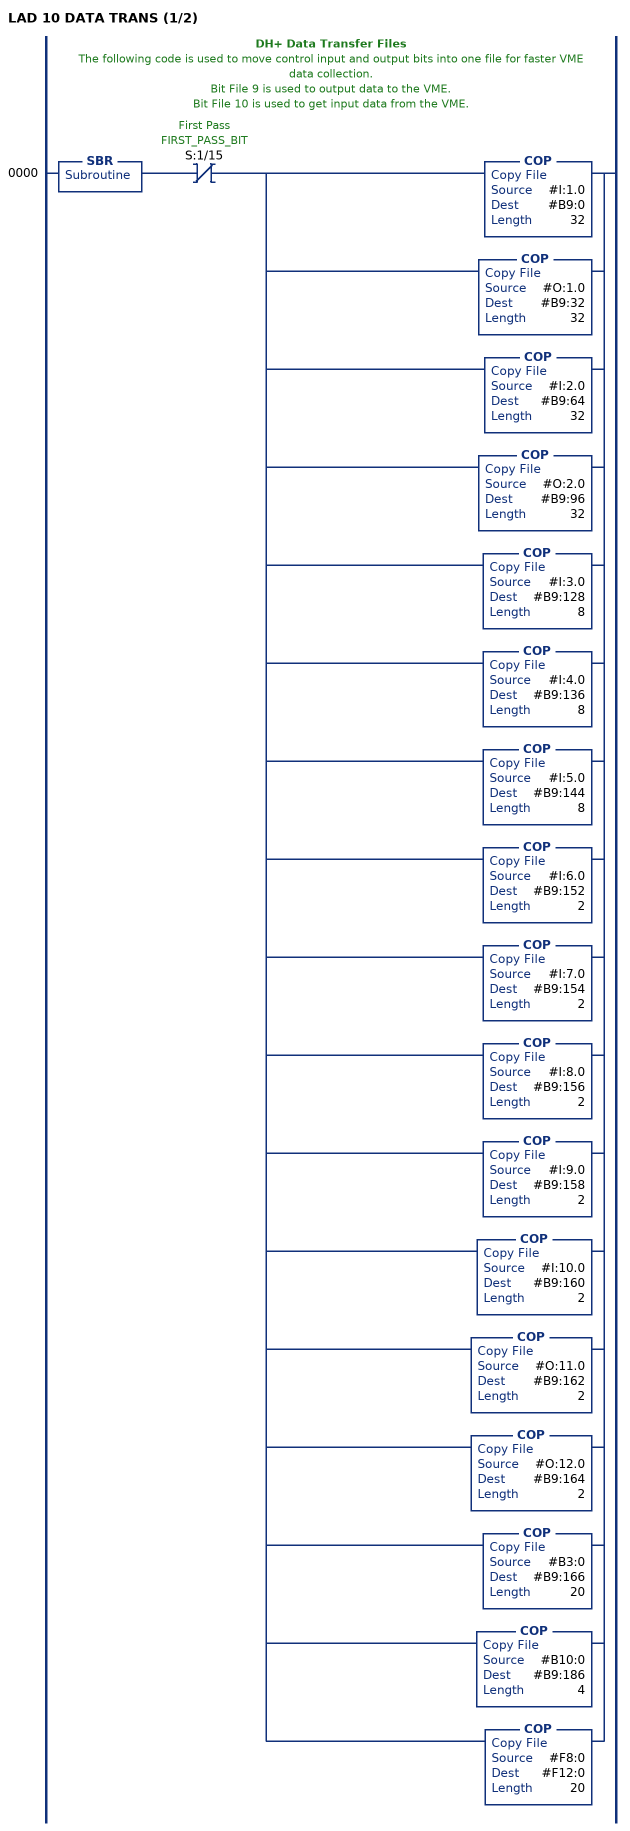
% Rung: 0 %
% TITLE: DH+ Data Transfer Files %
% The following code is used to move control input and output bits into one file for faster VME data collection.
% 
% 
% Bit File 9 is used to output data to the VME.
% 
% Bit File 10 is used to get input data from the VME. %
SOR SBR XIO S:1/15 BST COP #I:1.0 #B9:0 32 NXB COP #O:1.0 #B9:32 32 NXB COP #I:2.0 #B9:64 32 NXB COP #O:2.0 #B9:96 32 NXB COP #I:3.0 #B9:128 8 NXB COP #I:4.0 #B9:136 8 NXB COP #I:5.0 #B9:144 8 NXB COP #I:6.0 #B9:152 2 NXB COP #I:7.0 #B9:154 2 NXB COP #I:8.0 #B9:156 2 NXB COP #I:9.0 #B9:158 2 NXB COP #I:10.0 #B9:160 2 NXB COP #O:11.0 #B9:162 2 NXB COP #O:12.0 #B9:164 2 NXB COP #B3:0 #B9:166 20 NXB COP #B10:0 #B9:186 4 NXB COP #F8:0 #F12:0 20 BND EOR
%   S:1/15  FIRST_PASS_BIT  "First Pass" %
%   I:2.0  DCM_1_STATUS_WORD  "Direct communications module 1 status word." %
%   I:3.0  AZ_1_VOLTAGE  "Azimuth motor 1 voltage." %
%   I:4.0  ALT_POSITION  "Altitude clinometer raw position value." %
%   I:5.0  COUNTERWEIGHT_1_POS  "Counterweight #1 string pot position value" %
%   F8:0  AZ_MTR_1_RES  "Azimuth motor 1 calculated resistance value. Used for motor overtemp interlock." %

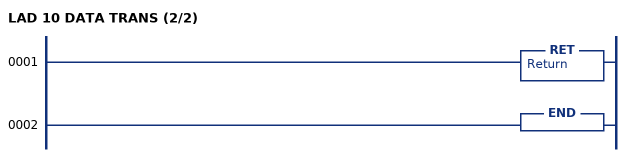
% Rung: 1 %
SOR RET EOR
% Rung: 2 %
SOR END EOR

LADDER 11 "BRAKE STOP"
